KUKA KRL program: MyProgram_163().src

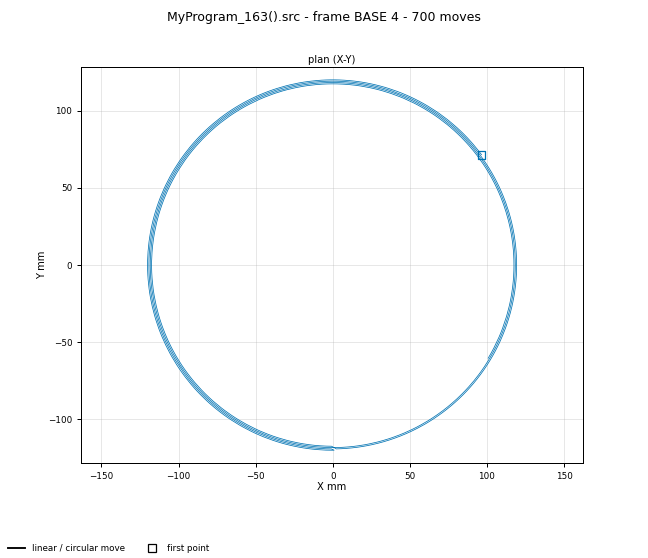
[picture p0: tool path of MyProgram_163().src in frame BASE 4, 700 of 700 moves have a stored position in this frame; points joined in program order, loops and branches not executed]
&ACCESS RVP
&REL 1
&PARAM TEMPLATE = C:\KRC\Roboter\Template\vorgabe
&PARAM EDITMASK = *
DEF MyProgram_163()
; ---- Setting reference (Base) ----
$BASE = BASE_DATA[4]

; --------------------------
; ---- Setting tool (TCP) ----
$TOOL = TOOL_DATA[3]
; --------------------------

$VEL.CP = VEL_APROX_PRINT
Startdeposition()
$VEL.CP = VEL_PRINT
LIN {X 96.4825,Y 71.5563,Z 124,A 32.763,B 24.9424,C -1.7531,E1 25.1279,E2 413.2714} C_DIS
LIN {X 94.5565,Y 74.0809,Z 124,A 34.1726,B 24.9424,C -1.7517,E1 25.1255,E2 411.8718} C_DIS
LIN {X 92.5032,Y 76.6279,Z 124,A 35.5868,B 24.9427,C -1.7484,E1 25.123,E2 410.4719} C_DIS
LIN {X 90.9571,Y 78.4601,Z 124,A 36.9601,B 24.9418,C -1.7622,E1 25.1205,E2 409.0724} C_DIS
LIN {X 89.0042,Y 80.6687,Z 124,A 38.3594,B 24.9416,C -1.7651,E1 25.1179,E2 407.6724} C_DIS
LIN {X 86.9977,Y 82.8287,Z 124,A 39.759,B 24.9414,C -1.7679,E1 25.1152,E2 406.2723} C_DIS
LIN {X 84.9388,Y 84.9388,Z 124,A 41.1588,B 24.9412,C -1.7707,E1 25.1124,E2 404.8719} C_DIS
LIN {X 82.8287,Y 86.9977,Z 124,A 42.5588,B 24.9411,C -1.7733,E1 25.1096,E2 403.4714} C_DIS
LIN {X 80.6687,Y 89.0042,Z 124,A 43.9588,B 24.9409,C -1.7759,E1 25.1067,E2 402.071} C_DIS
LIN {X 78.115,Y 91.2511,Z 124,A 45.38,B 24.9413,C -1.7695,E1 25.1038,E2 400.6704} C_DIS
LIN {X 76.2043,Y 92.8552,Z 124,A 46.7595,B 24.9406,C -1.7809,E1 25.1008,E2 399.2694} C_DIS
LIN {X 73.9026,Y 94.6974,Z 124,A 48.1603,B 24.9404,C -1.7832,E1 25.0977,E2 397.8683} C_DIS
LIN {X 71.2616,Y 96.6983,Z 124,A 49.578,B 24.9407,C -1.7783,E1 25.0946,E2 396.4673} C_DIS
LIN {X 69.167,Y 98.2096,Z 124,A 50.9622,B 24.9401,C -1.7877,E1 25.0914,E2 395.0657} C_DIS
LIN {X 66.736,Y 99.8774,Z 124,A 52.3632,B 24.94,C -1.7898,E1 25.0881,E2 393.6645} C_DIS
LIN {X 63.9427,Y 101.6863,Z 124,A 53.7826,B 24.9403,C -1.7844,E1 25.0849,E2 392.2626} C_DIS
LIN {X 61.7548,Y 103.0317,Z 124,A 55.2287,B 24.9395,C -1.7967,E1 25.0813,E2 390.7918} C_DIS
LIN {X 59.2077,Y 104.5162,Z 124,A 56.5684,B 24.9395,C -1.7956,E1 25.0781,E2 389.4588} C_DIS
LIN {X 56.1374,Y 106.1945,Z 124,A 58.2703,B 24.9393,C -1.7995,E1 25.0739,E2 387.7527} C_DIS
LIN {X 53.3205,Y 107.6363,Z 124,A 59.7249,B 24.9393,C -1.7988,E1 25.0703,E2 386.3035} C_DIS
LIN {X 50.7178,Y 108.8868,Z 124,A 61.1244,B 24.9392,C -1.8015,E1 25.0668,E2 384.9011} C_DIS
LIN {X 47.8151,Y 110.1926,Z 124,A 62.6869,B 24.9389,C -1.8054,E1 25.0628,E2 383.3335} C_DIS
LIN {X 44.6032,Y 111.5336,Z 124,A 64.2825,B 24.9389,C -1.804,E1 25.0586,E2 381.7446} C_DIS
LIN {X 41.8526,Y 112.5946,Z 124,A 65.6861,B 24.9389,C -1.8053,E1 25.055,E2 380.3411} C_DIS
LIN {X 38.6209,Y 113.7415,Z 124,A 67.1118,B 24.9395,C -1.7969,E1 25.0513,E2 378.938} C_DIS
LIN {X 36.2774,Y 114.5126,Z 124,A 68.4935,B 24.9388,C -1.8074,E1 25.0476,E2 377.5341} C_DIS
LIN {X 33.4562,Y 115.3684,Z 124,A 69.8975,B 24.9388,C -1.8084,E1 25.0438,E2 376.1303} C_DIS
LIN {X 30.6149,Y 116.1547,Z 124,A 71.3016,B 24.9386,C -1.8092,E1 25.04,E2 374.7265} C_DIS
LIN {X 27.7551,Y 116.871,Z 124,A 72.706,B 24.9386,C -1.8099,E1 25.0362,E2 373.3223} C_DIS
LIN {X 24.8785,Y 117.517,Z 124,A 74.1109,B 24.9386,C -1.8106,E1 25.0324,E2 371.9177} C_DIS
LIN {X 21.987,Y 118.0921,Z 124,A 75.5159,B 24.9386,C -1.8111,E1 25.0285,E2 370.5132} C_DIS
LIN {X 19.0823,Y 118.5962,Z 124,A 76.9212,B 24.9385,C -1.8116,E1 25.0246,E2 369.1082} C_DIS
LIN {X 16.166,Y 119.0288,Z 124,A 78.3267,B 24.9385,C -1.8119,E1 25.0208,E2 367.7032} C_DIS
LIN {X 13.2401,Y 119.3896,Z 124,A 79.7322,B 24.9385,C -1.8121,E1 25.0169,E2 366.2981} C_DIS
LIN {X 10.3061,Y 119.6786,Z 124,A 81.1409,B 24.9385,C -1.8124,E1 25.0129,E2 364.8897} C_DIS
LIN {X 7.3659,Y 119.8955,Z 124,A 82.5443,B 24.9385,C -1.8123,E1 25.009,E2 363.4871} C_DIS
LIN {X 4.4213,Y 120.0402,Z 124,A 83.951,B 24.9385,C -1.8123,E1 25.0051,E2 362.081} C_DIS
LIN {X 1.4741,Y 120.1125,Z 124,A 85.3576,B 24.9385,C -1.812,E1 25.0012,E2 360.675} C_DIS
LIN {X -1.4741,Y 120.1125,Z 124,A 86.7645,B 24.9385,C -1.8118,E1 24.9973,E2 359.2688} C_DIS
LIN {X -4.4213,Y 120.0402,Z 124,A 88.1715,B 24.9385,C -1.8114,E1 24.9933,E2 357.8624} C_DIS
LIN {X -7.3659,Y 119.8955,Z 124,A 89.579,B 24.9385,C -1.8109,E1 24.9894,E2 356.4557} C_DIS
LIN {X -10.3061,Y 119.6786,Z 124,A 90.9865,B 24.9385,C -1.8103,E1 24.9855,E2 355.0489} C_DIS
LIN {X -13.6363,Y 119.3432,Z 124,A 92.4129,B 24.9391,C -1.8018,E1 24.9816,E2 353.6419} C_DIS
LIN {X -16.166,Y 119.0288,Z 124,A 93.8336,B 24.9386,C -1.8103,E1 24.9776,E2 352.2001} C_DIS
LIN {X -19.0823,Y 118.5962,Z 124,A 95.2109,B 24.9387,C -1.808,E1 24.9738,E2 350.827} C_DIS
LIN {X -21.987,Y 118.0921,Z 124,A 96.6192,B 24.9387,C -1.807,E1 24.9699,E2 349.4196} C_DIS
LIN {X -25.3754,Y 117.4086,Z 124,A 98.0519,B 24.9395,C -1.796,E1 24.9661,E2 348.0114} C_DIS
LIN {X -27.7551,Y 116.8711,Z 124,A 99.4372,B 24.9389,C -1.8048,E1 24.9623,E2 346.6034} C_DIS
LIN {X -30.6149,Y 116.1547,Z 124,A 100.8465,B 24.939,C -1.8035,E1 24.9585,E2 345.1951} C_DIS
LIN {X -33.6095,Y 115.3229,Z 124,A 102.2635,B 24.9393,C -1.799,E1 24.9547,E2 343.7865} C_DIS
LIN {X -36.2774,Y 114.5126,Z 124,A 103.6656,B 24.9393,C -1.8007,E1 24.9509,E2 342.378} C_DIS
LIN {X -39.0768,Y 113.5878,Z 124,A 105.0757,B 24.9393,C -1.7991,E1 24.9472,E2 340.969} C_DIS
LIN {X -41.8526,Y 112.5946,Z 124,A 106.4858,B 24.9394,C -1.7974,E1 24.9435,E2 339.5599} C_DIS
LIN {X -44.6032,Y 111.5336,Z 124,A 107.8963,B 24.9396,C -1.7957,E1 24.9398,E2 338.1506} C_DIS
LIN {X -47.3269,Y 110.4054,Z 124,A 109.3068,B 24.9396,C -1.7938,E1 24.9362,E2 336.7411} C_DIS
LIN {X -50.0222,Y 109.2107,Z 124,A 110.7178,B 24.9398,C -1.7919,E1 24.9326,E2 335.3313} C_DIS
LIN {X -52.6873,Y 107.9502,Z 124,A 112.2257,B 24.9397,C -1.7942,E1 24.9288,E2 333.8142} C_DIS
LIN {X -55.3206,Y 106.6246,Z 124,A 113.6672,B 24.9397,C -1.7934,E1 24.9252,E2 332.3707} C_DIS
LIN {X -57.9207,Y 105.2349,Z 124,A 114.9515,B 24.9402,C -1.7856,E1 24.9221,E2 331.1013} C_DIS
LIN {X -60.4858,Y 103.7818,Z 124,A 116.3632,B 24.9404,C -1.7833,E1 24.9187,E2 329.6908} C_DIS
LIN {X -63.0145,Y 102.2661,Z 124,A 117.775,B 24.9406,C -1.7809,E1 24.9153,E2 328.2803} C_DIS
LIN {X -65.5053,Y 100.6888,Z 124,A 119.1871,B 24.9407,C -1.7785,E1 24.912,E2 326.8695} C_DIS
LIN {X -67.9566,Y 99.0509,Z 124,A 120.5993,B 24.9409,C -1.7759,E1 24.9087,E2 325.4587} C_DIS
LIN {X -70.3669,Y 97.3534,Z 124,A 122.1858,B 24.9406,C -1.7809,E1 24.9051,E2 323.8548} C_DIS
LIN {X -73.2948,Y 95.1658,Z 124,A 123.7761,B 24.9412,C -1.7706,E1 24.9016,E2 322.2833} C_DIS
LIN {X -75.6552,Y 93.3002,Z 124,A 125.192,B 24.9415,C -1.7666,E1 24.8985,E2 320.8717} C_DIS
LIN {X -77.876,Y 91.4547,Z 124,A 126.5891,B 24.9417,C -1.7643,E1 24.8955,E2 319.4745} C_DIS
LIN {X -80.097,Y 89.516,Z 124,A 128.0021,B 24.9419,C -1.7614,E1 24.8926,E2 318.0629} C_DIS
LIN {X -82.2697,Y 87.5234,Z 124,A 129.4156,B 24.9421,C -1.7584,E1 24.8897,E2 316.6508} C_DIS
LIN {X -84.3928,Y 85.478,Z 124,A 130.829,B 24.9423,C -1.7553,E1 24.8869,E2 315.2388} C_DIS
LIN {X -86.4652,Y 83.3812,Z 124,A 132.2427,B 24.9425,C -1.7521,E1 24.8841,E2 313.8266} C_DIS
LIN {X -88.4854,Y 81.2341,Z 124,A 133.67,B 24.9426,C -1.7495,E1 24.8814,E2 312.3993} C_DIS
LIN {X -90.4523,Y 79.0381,Z 124,A 135.0707,B 24.9429,C -1.7456,E1 24.8788,E2 311.0016} C_DIS
LIN {X -92.4035,Y 76.7479,Z 124,A 136.5141,B 24.9431,C -1.7422,E1 24.8762,E2 309.5596} C_DIS
LIN {X -94.2592,Y 74.4571,Z 124,A 137.9284,B 24.9433,C -1.7388,E1 24.8738,E2 308.1468} C_DIS
LIN {X -96.0216,Y 72.1698,Z 124,A 139.3138,B 24.9436,C -1.7354,E1 24.8714,E2 306.7629} C_DIS
LIN {X -97.7639,Y 69.7916,Z 124,A 140.7284,B 24.9438,C -1.7319,E1 24.8691,E2 305.3498} C_DIS
LIN {X -99.4472,Y 67.3714,Z 124,A 142.1433,B 24.944,C -1.7283,E1 24.8669,E2 303.9364} C_DIS
LIN {X -101.1378,Y 64.8058,Z 124,A 143.605,B 24.9443,C -1.724,E1 24.8647,E2 302.4776} C_DIS
LIN {X -102.6662,Y 62.3562,Z 124,A 145.003,B 24.9445,C -1.7209,E1 24.8626,E2 301.0798} C_DIS
LIN {X -104.1641,Y 59.8205,Z 124,A 146.4171,B 24.9447,C -1.7172,E1 24.8606,E2 299.6672} C_DIS
LIN {X -105.6008,Y 57.2461,Z 124,A 147.819,B 24.945,C -1.7129,E1 24.8588,E2 298.2683} C_DIS
LIN {X -107.0122,Y 54.5623,Z 124,A 149.2718,B 24.9453,C -1.7088,E1 24.8569,E2 296.8174} C_DIS
LIN {X -108.2825,Y 51.9956,Z 124,A 150.6629,B 24.9455,C -1.7058,E1 24.8552,E2 295.426} C_DIS
LIN {X -109.5259,Y 49.3226,Z 124,A 152.0655,B 24.9458,C -1.7013,E1 24.8536,E2 294.0263} C_DIS
LIN {X -110.7034,Y 46.6198,Z 124,A 153.4938,B 24.946,C -1.698,E1 24.852,E2 292.5981} C_DIS
LIN {X -111.792,Y 43.9454,Z 124,A 154.8937,B 24.9462,C -1.6946,E1 24.8505,E2 291.1984} C_DIS
LIN {X -112.8576,Y 41.1317,Z 124,A 156.3363,B 24.9464,C -1.6905,E1 24.8491,E2 289.7576} C_DIS
LIN {X -113.8851,Y 38.1951,Z 124,A 157.883,B 24.9466,C -1.6885,E1 24.8477,E2 288.2068} C_DIS
LIN {X -114.9492,Y 34.8694,Z 124,A 159.4964,B 24.9471,C -1.6809,E1 24.8464,E2 286.6022} C_DIS
LIN {X -115.7703,Y 32.0379,Z 124,A 160.9124,B 24.9473,C -1.6768,E1 24.8453,E2 285.1876} C_DIS
LIN {X -116.5217,Y 29.1872,Z 124,A 162.3285,B 24.9476,C -1.6727,E1 24.8444,E2 283.7731} C_DIS
LIN {X -117.2029,Y 26.3188,Z 124,A 163.7444,B 24.9478,C -1.6686,E1 24.8435,E2 282.3587} C_DIS
LIN {X -117.8134,Y 23.4345,Z 124,A 165.1604,B 24.9481,C -1.6645,E1 24.8427,E2 280.9441} C_DIS
LIN {X -118.3531,Y 20.5362,Z 124,A 166.5765,B 24.9483,C -1.6604,E1 24.842,E2 279.5296} C_DIS
LIN {X -118.8214,Y 17.6255,Z 124,A 167.9925,B 24.9486,C -1.6562,E1 24.8414,E2 278.1151} C_DIS
LIN {X -119.2182,Y 14.7042,Z 124,A 169.4089,B 24.9489,C -1.652,E1 24.8409,E2 276.7001} C_DIS
LIN {X -119.5529,Y 11.6682,Z 124,A 170.8298,B 24.9492,C -1.6458,E1 24.8405,E2 275.2856} C_DIS
LIN {X -119.7961,Y 8.8367,Z 124,A 172.241,B 24.9494,C -1.6437,E1 24.8401,E2 273.8709} C_DIS
LIN {X -119.9855,Y 5.6936,Z 124,A 173.6666,B 24.9499,C -1.6356,E1 24.8399,E2 272.4561} C_DIS
LIN {X -120.0854,Y 2.9479,Z 124,A 175.0732,B 24.9499,C -1.6354,E1 24.8399,E2 271.0415} C_DIS
LIN {X -120.1192,Y -0.4835,Z 124,A 176.796,B 24.9499,C -1.6337,E1 24.8398,E2 269.3123} C_DIS
LIN {X -120.0637,Y -3.6544,Z 124,A 178.245,B 24.9505,C -1.6261,E1 24.8398,E2 267.8727} C_DIS
LIN {X -119.9378,Y -6.5998,Z 124,A 179.6742,B 24.9507,C -1.6225,E1 24.8401,E2 266.4435} C_DIS
LIN {X -119.7398,Y -9.5412,Z 124,A -178.9099,B 24.9509,C -1.6184,E1 24.8404,E2 265.0289} C_DIS
LIN {X -119.4632,Y -12.5371,Z 124,A -177.491,B 24.9512,C -1.613,E1 24.8408,E2 263.6141} C_DIS
LIN {X -119.1274,Y -15.4051,Z 124,A -176.0777,B 24.9514,C -1.6101,E1 24.8413,E2 262.1993} C_DIS
LIN {X -118.7042,Y -18.3838,Z 124,A -174.646,B 24.9517,C -1.6054,E1 24.8418,E2 260.7704} C_DIS
LIN {X -118.2172,Y -21.2914,Z 124,A -173.2434,B 24.952,C -1.6008,E1 24.8425,E2 259.3704} C_DIS
LIN {X -117.6591,Y -24.1862,Z 124,A -171.8273,B 24.9522,C -1.5968,E1 24.8433,E2 257.9556} C_DIS
LIN {X -117.0438,Y -27.0074,Z 124,A -170.4277,B 24.9524,C -1.5934,E1 24.8441,E2 256.5557} C_DIS
LIN {X -116.3306,Y -29.9303,Z 124,A -168.996,B 24.9527,C -1.5888,E1 24.8451,E2 255.1266} C_DIS
LIN {X -115.5776,Y -32.7179,Z 124,A -167.5966,B 24.9529,C -1.5855,E1 24.8462,E2 253.7271} C_DIS
LIN {X -114.7398,Y -35.5445,Z 124,A -166.1679,B 24.9531,C -1.5822,E1 24.8473,E2 252.2981} C_DIS
LIN {X -113.8136,Y -38.4071,Z 124,A -164.7495,B 24.9534,C -1.5771,E1 24.8486,E2 250.8836} C_DIS
LIN {X -112.8576,Y -41.1317,Z 124,A -163.3371,B 24.9536,C -1.5745,E1 24.8499,E2 249.4695} C_DIS
LIN {X -111.792,Y -43.9454,Z 124,A -161.9058,B 24.9538,C -1.5701,E1 24.8513,E2 248.0406} C_DIS
LIN {X -110.6798,Y -46.6756,Z 124,A -160.4908,B 24.954,C -1.5663,E1 24.8528,E2 246.6267} C_DIS
LIN {X -109.501,Y -49.3778,Z 124,A -159.089,B 24.9543,C -1.5621,E1 24.8544,E2 245.2274} C_DIS
LIN {X -108.2825,Y -51.9956,Z 124,A -157.69,B 24.9545,C -1.5591,E1 24.8561,E2 243.8278} C_DIS
LIN {X -106.9458,Y -54.6923,Z 124,A -156.2588,B 24.9547,C -1.5548,E1 24.8579,E2 242.3991} C_DIS
LIN {X -105.6008,Y -57.2462,Z 124,A -154.8475,B 24.9548,C -1.5525,E1 24.8598,E2 240.9858} C_DIS
LIN {X -104.1641,Y -59.8205,Z 124,A -153.4461,B 24.9551,C -1.5485,E1 24.8617,E2 239.5868} C_DIS
LIN {X -102.6332,Y -62.4106,Z 124,A -152.0026,B 24.9553,C -1.545,E1 24.8638,E2 238.1441} C_DIS
LIN {X -101.1033,Y -64.8595,Z 124,A -150.6177,B 24.9555,C -1.5417,E1 24.8658,E2 236.7601} C_DIS
LIN {X -99.4472,Y -67.3714,Z 124,A -149.1742,B 24.9557,C -1.5383,E1 24.8681,E2 235.3173} C_DIS
LIN {X -97.6554,Y -69.9437,Z 124,A -147.6122,B 24.9557,C -1.5374,E1 24.8706,E2 233.7498} C_DIS
LIN {X -95.5972,Y -72.7349,Z 124,A -146.0079,B 24.9561,C -1.5311,E1 24.8733,E2 232.1528} C_DIS
LIN {X -93.6748,Y -75.193,Z 124,A -144.5862,B 24.9565,C -1.5246,E1 24.8757,E2 230.7398} C_DIS
LIN {X -91.9131,Y -77.338,Z 124,A -143.1807,B 24.9565,C -1.525,E1 24.8782,E2 229.3269} C_DIS
LIN {X -89.9874,Y -79.5704,Z 124,A -141.7676,B 24.9565,C -1.5221,E1 24.8808,E2 227.9145} C_DIS
LIN {X -88.0076,Y -81.7548,Z 124,A -140.3545,B 24.9568,C -1.5192,E1 24.8835,E2 226.5019} C_DIS
LIN {X -85.9747,Y -83.89,Z 124,A -138.9417,B 24.9569,C -1.5164,E1 24.8862,E2 225.0896} C_DIS
LIN {X -83.8593,Y -86.0043,Z 124,A -137.527,B 24.9571,C -1.5129,E1 24.889,E2 223.6775} C_DIS
LIN {X -81.7548,Y -88.0076,Z 124,A -136.1165,B 24.9572,C -1.5111,E1 24.8919,E2 222.2654} C_DIS
LIN {X -79.5704,Y -89.9874,Z 124,A -134.6582,B 24.9572,C -1.5106,E1 24.895,E2 220.8026} C_DIS
LIN {X -77.338,Y -91.9131,Z 124,A -133.2919,B 24.9575,C -1.5061,E1 24.8979,E2 219.4417} C_DIS
LIN {X -75.0591,Y -93.7834,Z 124,A -131.7279,B 24.9573,C -1.5105,E1 24.9013,E2 217.8614} C_DIS
LIN {X -72.7349,Y -95.5972,Z 124,A -130.4684,B 24.9578,C -1.5014,E1 24.904,E2 216.6189} C_DIS
LIN {X -70.3669,Y -97.3534,Z 124,A -129.057,B 24.9578,C -1.4992,E1 24.9072,E2 215.2078} C_DIS
LIN {X -67.9566,Y -99.0509,Z 124,A -127.4996,B 24.9576,C -1.5036,E1 24.9108,E2 213.6346} C_DIS
LIN {X -65.5053,Y -100.6888,Z 124,A -126.2346,B 24.9581,C -1.495,E1 24.9137,E2 212.386} C_DIS
LIN {X -62.8141,Y -102.3879,Z 124,A -124.8127,B 24.9585,C -1.4884,E1 24.9171,E2 210.9753} C_DIS
LIN {X -60.4858,Y -103.7818,Z 124,A -123.2395,B 24.9579,C -1.499,E1 24.9209,E2 209.3721} C_DIS
LIN {X -57.9207,Y -105.2349,Z 124,A -122.0025,B 24.9584,C -1.4894,E1 24.9239,E2 208.1543} C_DIS
LIN {X -54.8467,Y -106.8669,Z 124,A -120.5673,B 24.9591,C -1.4771,E1 24.9274,E2 206.7443} C_DIS
LIN {X -52.6873,Y -107.9502,Z 124,A -119.1824,B 24.9586,C -1.4861,E1 24.9309,E2 205.3343} C_DIS
LIN {X -50.0222,Y -109.2107,Z 124,A -117.7726,B 24.9587,C -1.4847,E1 24.9345,E2 203.9246} C_DIS
LIN {X -47.3269,Y -110.4054,Z 124,A -116.363,B 24.9587,C -1.4833,E1 24.9381,E2 202.5149} C_DIS
LIN {X -44.6032,Y -111.5336,Z 124,A -114.9061,B 24.9587,C -1.4842,E1 24.9419,E2 201.0526} C_DIS
LIN {X -41.6064,Y -112.6844,Z 124,A -113.5323,B 24.9592,C -1.4756,E1 24.9454,E2 199.6964} C_DIS
LIN {X -39.0768,Y -113.5878,Z 124,A -112.1361,B 24.959,C -1.4797,E1 24.9491,E2 198.2876} C_DIS
LIN {X -36.2774,Y -114.5126,Z 124,A -110.7272,B 24.959,C -1.4787,E1 24.9529,E2 196.8785} C_DIS
LIN {X -33.4562,Y -115.3684,Z 124,A -109.3189,B 24.959,C -1.4778,E1 24.9567,E2 195.47} C_DIS
LIN {X -30.6149,Y -116.1547,Z 124,A -107.9109,B 24.9591,C -1.477,E1 24.9605,E2 194.0618} C_DIS
LIN {X -27.7551,Y -116.8711,Z 124,A -106.502,B 24.9591,C -1.4764,E1 24.9643,E2 192.6524} C_DIS
LIN {X -24.8785,Y -117.517,Z 124,A -105.0952,B 24.9592,C -1.4757,E1 24.9681,E2 191.2455} C_DIS
LIN {X -21.987,Y -118.0921,Z 124,A -103.6879,B 24.9592,C -1.4752,E1 24.972,E2 189.8378} C_DIS
LIN {X -19.0823,Y -118.5962,Z 124,A -102.2806,B 24.9592,C -1.4748,E1 24.9759,E2 188.43} C_DIS
LIN {X -16.166,Y -119.0288,Z 124,A -100.8736,B 24.9592,C -1.4746,E1 24.9798,E2 187.0226} C_DIS
LIN {X -13.2401,Y -119.3896,Z 124,A -99.4671,B 24.9592,C -1.4744,E1 24.9837,E2 185.6156} C_DIS
LIN {X -10.3061,Y -119.6786,Z 124,A -98.0605,B 24.9592,C -1.4743,E1 24.9876,E2 184.2085} C_DIS
LIN {X -7.1561,Y -119.9071,Z 124,A -96.4549,B 24.959,C -1.479,E1 24.9921,E2 182.5913} C_DIS
LIN {X -4.4213,Y -120.0402,Z 124,A -95.2482,B 24.9593,C -1.4744,E1 24.9954,E2 181.395} C_DIS
LIN {X -1.4741,Y -120.1125,Z 124,A -93.8425,B 24.9593,C -1.4746,E1 24.9993,E2 179.9888} C_DIS
LIN {X 0.8495,Y -120.1163,Z 124,A -93.0999,B 24.9602,C -1.4579,E1 25.0013,E2 179.2859} C_DIS
Enddeposition()
LIN {X 0.8495,Y -120.1163,Z 124,A -93.0999,B 24.9602,C -1.4579,E1 25.0013,E2 179.2859} C_DIS
Startdeposition()
$VEL.CP = VEL_PRINT
LIN {X -0.9086,Y -119.2481,Z 124,A -94.2495,B 24.9602,C -1.4589,E1 24.9981,E2 180.4331} C_DIS
LIN {X -4.3095,Y -119.1753,Z 124,A -96.1957,B 24.9609,C -1.4444,E1 24.9926,E2 182.4138} C_DIS
LIN {X -10.5482,Y -118.7847,Z 124,A -98.7422,B 24.9598,C -1.4652,E1 24.9856,E2 184.912} C_DIS
LIN {X -13.5113,Y -118.4841,Z 124,A -100.4433,B 24.9604,C -1.4531,E1 24.9808,E2 186.6429} C_DIS
LIN {X -17.3471,Y -117.9844,Z 124,A -102.2953,B 24.9604,C -1.4538,E1 24.9757,E2 188.4946} C_DIS
LIN {X -21.1648,Y -117.3582,Z 124,A -104.0505,B 24.9601,C -1.4591,E1 24.9709,E2 190.239} C_DIS
LIN {X -24.6012,Y -116.6879,Z 124,A -105.8898,B 24.9605,C -1.4527,E1 24.9658,E2 192.0956} C_DIS
LIN {X -28.42,Y -115.8155,Z 124,A -107.6525,B 24.9601,C -1.4591,E1 24.961,E2 193.8456} C_DIS
LIN {X -31.8672,Y -114.9166,Z 124,A -109.4755,B 24.9603,C -1.4552,E1 24.9561,E2 195.6806} C_DIS
LIN {X -35.357,Y -113.8893,Z 124,A -111.1658,B 24.9601,C -1.459,E1 24.9516,E2 197.3647} C_DIS
LIN {X -38.8928,Y -112.7326,Z 124,A -113.0518,B 24.9603,C -1.4561,E1 24.9466,E2 199.2611} C_DIS
LIN {X -42.3587,Y -111.4749,Z 124,A -115.882,B 24.9627,C -1.4114,E1 24.939,E2 202.2035} C_DIS
LIN {X -49.0255,Y -108.7078,Z 124,A -118.1271,B 24.9596,C -1.4686,E1 24.9335,E2 204.318} C_DIS
LIN {X -51.8005,Y -107.4134,Z 124,A -119.6389,B 24.9596,C -1.4686,E1 24.9297,E2 205.8337} C_DIS
LIN {X -55.2299,Y -105.6915,Z 124,A -121.5594,B 24.9596,C -1.4676,E1 24.9249,E2 207.7618} C_DIS
LIN {X -58.4356,Y -103.9533,Z 124,A -123.338,B 24.9596,C -1.4688,E1 24.9205,E2 209.5426} C_DIS
LIN {X -62.5813,Y -101.5134,Z 124,A -125.6725,B 24.9595,C -1.4712,E1 24.9149,E2 211.8786} C_DIS
LIN {X -65.6775,Y -99.5357,Z 124,A -127.3041,B 24.959,C -1.4799,E1 24.9112,E2 213.4948} C_DIS
LIN {X -68.6467,Y -97.5142,Z 124,A -129.1599,B 24.9591,C -1.4771,E1 24.9069,E2 215.3636} C_DIS
LIN {X -72.1893,Y -94.9214,Z 124,A -131.119,B 24.9586,C -1.4873,E1 24.9025,E2 217.3053} C_DIS
LIN {X -74.6388,Y -93.0068,Z 124,A -133.1968,B 24.9598,C -1.4649,E1 24.8979,E2 219.4442} C_DIS
LIN {X -77.7841,Y -90.3929,Z 124,A -134.4988,B 24.958,C -1.4973,E1 24.8952,E2 220.6742} C_DIS
LIN {X -81.2747,Y -87.2677,Z 124,A -136.942,B 24.9582,C -1.4935,E1 24.8901,E2 223.1362} C_DIS
LIN {X -83.8457,Y -84.7986,Z 124,A -138.6371,B 24.958,C -1.4979,E1 24.8867,E2 224.8279} C_DIS
LIN {X -86.3311,Y -82.2697,Z 124,A -140.4782,B 24.958,C -1.4957,E1 24.8832,E2 226.6822} C_DIS
LIN {X -89.3008,Y -79.0362,Z 124,A -142.4251,B 24.9574,C -1.5075,E1 24.8795,E2 228.6097} C_DIS
LIN {X -91.7598,Y -76.1645,Z 124,A -144.3636,B 24.9574,C -1.5065,E1 24.876,E2 230.5593} C_DIS
LIN {X -94.2396,Y -73.0747,Z 124,A -146.2329,B 24.9571,C -1.5126,E1 24.8728,E2 232.4231} C_DIS
LIN {X -96.7104,Y -69.7738,Z 124,A -148.275,B 24.9571,C -1.5149,E1 24.8694,E2 234.4695} C_DIS
LIN {X -101.6426,Y -62.3693,Z 124,A -152.3443,B 24.9559,C -1.5347,E1 24.8632,E2 238.5119} C_DIS
LIN {X -103.5586,Y -59.1322,Z 124,A -154.3041,B 24.9559,C -1.5332,E1 24.8604,E2 240.4857} C_DIS
LIN {X -105.8623,Y -54.9051,Z 124,A -156.5785,B 24.9555,C -1.5412,E1 24.8574,E2 242.753} C_DIS
LIN {X -107.973,Y -50.6244,Z 124,A -159.2947,B 24.9561,C -1.5299,E1 24.8541,E2 245.5108} C_DIS
LIN {X -109.3185,Y -47.6483,Z 124,A -160.5271,B 24.9551,C -1.5486,E1 24.8528,E2 246.7055} C_DIS
LIN {X -110.7063,Y -44.3336,Z 124,A -162.3317,B 24.955,C -1.5504,E1 24.8508,E2 248.5159} C_DIS
LIN {X -112.0876,Y -40.7099,Z 124,A -164.1388,B 24.9545,C -1.5583,E1 24.8491,E2 250.3143} C_DIS
LIN {X -113.3767,Y -36.9688,Z 124,A -166.0891,B 24.9543,C -1.562,E1 24.8473,E2 252.2669} C_DIS
LIN {X -114.3673,Y -33.7793,Z 124,A -167.594,B 24.9538,C -1.5711,E1 24.8461,E2 253.7589} C_DIS
LIN {X -115.2284,Y -30.7158,Z 124,A -169.5376,B 24.9545,C -1.5585,E1 24.8447,E2 255.7437} C_DIS
LIN {X -116.0384,Y -27.5037,Z 124,A -170.7328,B 24.9532,C -1.5799,E1 24.8439,E2 256.8948} C_DIS
LIN {X -116.7334,Y -24.3797,Z 124,A -172.4192,B 24.9533,C -1.5786,E1 24.8429,E2 258.5944} C_DIS
LIN {X -117.4761,Y -20.5095,Z 124,A -174.4096,B 24.9532,C -1.5805,E1 24.8419,E2 260.592} C_DIS
LIN {X -118.0541,Y -16.8565,Z 124,A -176.0713,B 24.9526,C -1.591,E1 24.8412,E2 262.2385} C_DIS
LIN {X -118.5456,Y -12.9668,Z 124,A -177.9811,B 24.9523,C -1.5959,E1 24.8406,E2 264.148} C_DIS
LIN {X -118.8944,Y -9.2243,Z 124,A -179.662,B 24.9516,C -1.607,E1 24.8402,E2 265.8126} C_DIS
LIN {X -119.1031,Y -5.9771,Z 124,A 178.7165,B 24.9515,C -1.6096,E1 24.8399,E2 267.4376} C_DIS
LIN {X -119.2222,Y -2.6833,Z 124,A 177.0032,B 24.9515,C -1.6094,E1 24.8399,E2 269.1617} C_DIS
LIN {X -119.2486,Y 0.8732,Z 124,A 175.3921,B 24.9509,C -1.619,E1 24.8398,E2 270.7596} C_DIS
LIN {X -119.1841,Y 4.0209,Z 124,A 173.7356,B 24.9509,C -1.618,E1 24.8399,E2 272.4286} C_DIS
LIN {X -118.9864,Y 7.9461,Z 124,A 171.9116,B 24.9504,C -1.6268,E1 24.8402,E2 274.2425} C_DIS
LIN {X -118.7073,Y 11.3863,Z 124,A 170.2503,B 24.9501,C -1.6321,E1 24.8406,E2 275.9012} C_DIS
LIN {X -118.3042,Y 15.0041,Z 124,A 168.4558,B 24.9499,C -1.6359,E1 24.8412,E2 277.6973} C_DIS
LIN {X -117.8441,Y 18.2666,Z 124,A 166.8664,B 24.9496,C -1.6408,E1 24.8419,E2 279.2844} C_DIS
LIN {X -117.0758,Y 22.6755,Z 124,A 164.6811,B 24.9492,C -1.6463,E1 24.843,E2 281.4696} C_DIS
LIN {X -115.8658,Y 28.2138,Z 124,A 162.0185,B 24.9485,C -1.6577,E1 24.8446,E2 284.1209} C_DIS
LIN {X -114.2551,Y 34.1576,Z 124,A 159.137,B 24.9477,C -1.6703,E1 24.8467,E2 286.9889} C_DIS
LIN {X -113.4175,Y 36.8427,Z 124,A 157.6393,B 24.9478,C -1.6685,E1 24.848,E2 288.4995} C_DIS
LIN {X -111.7902,Y 41.5218,Z 124,A 154.9447,B 24.9482,C -1.6629,E1 24.8506,E2 291.2227} C_DIS
LIN {X -109.7259,Y 46.7045,Z 124,A 152.5464,B 24.9469,C -1.6829,E1 24.8531,E2 293.5867} C_DIS
LIN {X -108.22,Y 50.0939,Z 124,A 150.7165,B 24.9467,C -1.6864,E1 24.8552,E2 295.4184} C_DIS
LIN {X -106.7333,Y 53.188,Z 124,A 149.1005,B 24.9463,C -1.6927,E1 24.8572,E2 297.028} C_DIS
LIN {X -104.4869,Y 57.4795,Z 124,A 146.5852,B 24.9463,C -1.6918,E1 24.8605,E2 299.5588} C_DIS
LIN {X -102.5854,Y 60.8043,Z 124,A 144.9339,B 24.9455,C -1.7051,E1 24.8628,E2 301.1871} C_DIS
LIN {X -100.6939,Y 63.8907,Z 124,A 143.0375,B 24.9456,C -1.7035,E1 24.8656,E2 303.0969} C_DIS
LIN {X -98.4349,Y 67.3184,Z 124,A 140.9981,B 24.9454,C -1.7062,E1 24.8688,E2 305.1399} C_DIS
LIN {X -96.4855,Y 70.0832,Z 124,A 139.6672,B 24.9444,C -1.7231,E1 24.8709,E2 306.4372} C_DIS
LIN {X -94.6769,Y 72.5073,Z 124,A 138.035,B 24.9446,C -1.7195,E1 24.8737,E2 308.0857} C_DIS
LIN {X -92.4248,Y 75.357,Z 124,A 136.3123,B 24.9442,C -1.7251,E1 24.8767,E2 309.8032} C_DIS
LIN {X -89.7308,Y 78.5449,Z 124,A 134.356,B 24.9438,C -1.7324,E1 24.8802,E2 311.751} C_DIS
LIN {X -85.7767,Y 82.8449,Z 124,A 131.4879,B 24.9435,C -1.7369,E1 24.8857,E2 314.621} C_DIS
LIN {X -83.1345,Y 85.4975,Z 124,A 129.4443,B 24.9439,C -1.7309,E1 24.8898,E2 316.6874} C_DIS
LIN {X -79.7203,Y 88.6883,Z 124,A 126.9343,B 24.9442,C -1.725,E1 24.895,E2 319.2215} C_DIS
LIN {X -76.7203,Y 91.298,Z 124,A 125.4167,B 24.9429,C -1.7459,E1 24.8982,E2 320.6953} C_DIS
LIN {X -73.8278,Y 93.6502,Z 124,A 123.6934,B 24.9424,C -1.7527,E1 24.9019,E2 322.4088} C_DIS
LIN {X -71.0064,Y 95.8095,Z 124,A 121.2018,B 24.9444,C -1.7231,E1 24.9077,E2 324.9796} C_DIS
LIN {X -66.7964,Y 98.7884,Z 124,A 119.6097,B 24.9416,C -1.7657,E1 24.9111,E2 326.4759} C_DIS
LIN {X -64.418,Y 100.3555,Z 124,A 118.1215,B 24.9417,C -1.7632,E1 24.9146,E2 327.9748} C_DIS
LIN {X -61.4782,Y 102.1842,Z 124,A 116.3527,B 24.9418,C -1.7618,E1 24.9188,E2 329.7525} C_DIS
LIN {X -56.5006,Y 105.0178,Z 124,A 114.0451,B 24.9402,C -1.7858,E1 24.9243,E2 332.0099} C_DIS
LIN {X -51.2487,Y 107.6785,Z 124,A 110.2878,B 24.9426,C -1.7504,E1 24.934,E2 335.8611} C_DIS
LIN {X -47.4136,Y 109.4208,Z 124,A 108.9596,B 24.9404,C -1.7833,E1 24.9372,E2 337.1142} C_DIS
LIN {X -44.8215,Y 110.5077,Z 124,A 107.5114,B 24.9405,C -1.781,E1 24.9409,E2 338.5711} C_DIS
LIN {X -41.7792,Y 111.6944,Z 124,A 105.6075,B 24.9414,C -1.7686,E1 24.946,E2 340.5085} C_DIS
LIN {X -36.7399,Y 113.4508,Z 124,A 103.3352,B 24.9403,C -1.7845,E1 24.9519,E2 342.7475} C_DIS
LIN {X -33.6255,Y 114.4129,Z 124,A 101.8139,B 24.9401,C -1.7882,E1 24.9559,E2 344.2626} C_DIS
LIN {X -29.33,Y 115.5889,Z 124,A 99.4968,B 24.9404,C -1.7826,E1 24.9622,E2 346.5963} C_DIS
LIN {X -25.0419,Y 116.5931,Z 124,A 97.5053,B 24.9399,C -1.79,E1 24.9676,E2 348.5729} C_DIS
LIN {X -21.6386,Y 117.273,Z 124,A 95.7571,B 24.9401,C -1.7878,E1 24.9724,E2 350.3282} C_DIS
LIN {X -18.1261,Y 117.8658,Z 124,A 94.0876,B 24.9399,C -1.7909,E1 24.977,E2 351.9919} C_DIS
LIN {X -14.6574,Y 118.3491,Z 124,A 92.433,B 24.9397,C -1.7931,E1 24.9816,E2 353.6424} C_DIS
LIN {X -11.1145,Y 118.7324,Z 124,A 90.6712,B 24.9398,C -1.7919,E1 24.9865,E2 355.4082} C_DIS
LIN {X -7.9101,Y 118.9888,Z 124,A 89.1459,B 24.9398,C -1.7934,E1 24.9907,E2 356.9305} C_DIS
LIN {X -4.7004,Y 119.1595,Z 124,A 87.514,B 24.9399,C -1.79,E1 24.9953,E2 358.5708} C_DIS
LIN {X -0.8136,Y 119.2486,Z 124,A 85.7804,B 24.9395,C -1.7965,E1 25.0001,E2 360.2892} C_DIS
LIN {X 2.4858,Y 119.2258,Z 124,A 84.201,B 24.9395,C -1.797,E1 25.0045,E2 361.8672} C_DIS
LIN {X 5.7686,Y 119.1136,Z 124,A 82.4794,B 24.9399,C -1.7906,E1 25.0094,E2 363.6034} C_DIS
LIN {X 9.5817,Y 118.8659,Z 124,A 80.7469,B 24.9396,C -1.7952,E1 25.0142,E2 365.3241} C_DIS
LIN {X 13.1484,Y 118.5266,Z 124,A 78.8933,B 24.94,C -1.789,E1 25.0193,E2 367.1913} C_DIS
LIN {X 16.9309,Y 118.0435,Z 124,A 77.2415,B 24.9395,C -1.7967,E1 25.0239,E2 368.8234} C_DIS
LIN {X 20.1074,Y 117.5448,Z 124,A 75.606,B 24.9398,C -1.7921,E1 25.0284,E2 370.4682} C_DIS
LIN {X 23.7661,Y 116.8594,Z 124,A 73.8254,B 24.9398,C -1.7917,E1 25.0333,E2 372.2477} C_DIS
LIN {X 26.7556,Y 116.2112,Z 124,A 72.368,B 24.9398,C -1.7915,E1 25.0372,E2 373.7036} C_DIS
LIN {X 30.2559,Y 115.3509,Z 124,A 70.6234,B 24.94,C -1.7898,E1 25.042,E2 375.4495} C_DIS
LIN {X 33.9813,Y 114.3074,Z 124,A 68.7544,B 24.94,C -1.788,E1 25.047,E2 377.3195} C_DIS
LIN {X 37.6754,Y 113.1444,Z 124,A 66.9235,B 24.94,C -1.7879,E1 25.0518,E2 379.1474} C_DIS
LIN {X 46.3321,Y 109.8828,Z 124,A 62.511,B 24.9403,C -1.7849,E1 25.0634,E2 383.5572} C_DIS
LIN {X 49.6004,Y 108.4488,Z 124,A 60.5576,B 24.9412,C -1.7719,E1 25.0684,E2 385.5365} C_DIS
LIN {X 53.8467,Y 106.4033,Z 124,A 58.505,B 24.9407,C -1.7789,E1 25.0735,E2 387.5673} C_DIS
LIN {X 56.8704,Y 104.8172,Z 124,A 56.8441,B 24.9409,C -1.7757,E1 25.0776,E2 389.2309} C_DIS
LIN {X 60.3043,Y 102.8809,Z 124,A 54.7179,B 24.9418,C -1.7622,E1 25.0828,E2 391.3827} C_DIS
LIN {X 65.142,Y 99.8888,Z 124,A 52.1625,B 24.9415,C -1.7661,E1 25.0887,E2 393.9206} C_DIS
LIN {X 68.939,Y 97.306,Z 124,A 50.0308,B 24.9415,C -1.7658,E1 25.0936,E2 396.0456} C_DIS
LIN {X 71.85,Y 95.1764,Z 124,A 48.3153,B 24.9417,C -1.7636,E1 25.0975,E2 397.7604} C_DIS
LIN {X 75.3333,Y 92.444,Z 124,A 46.3141,B 24.9416,C -1.7655,E1 25.1018,E2 399.7495} C_DIS
LIN {X 77.7251,Y 90.4431,Z 124,A 44.7049,B 24.9421,C -1.7573,E1 25.1053,E2 401.3718} C_DIS
LIN {X 80.568,Y 87.9187,Z 124,A 42.9215,B 24.9422,C -1.7557,E1 25.109,E2 403.152} C_DIS
LIN {X 82.9768,Y 85.6495,Z 124,A 41.3149,B 24.9425,C -1.7515,E1 25.1122,E2 404.7617} C_DIS
LIN {X 85.7538,Y 82.8686,Z 124,A 39.4641,B 24.9427,C -1.7492,E1 25.1158,E2 406.6101} C_DIS
LIN {X 88.1066,Y 80.3633,Z 124,A 37.8299,B 24.9428,C -1.7462,E1 25.1189,E2 408.244} C_DIS
LIN {X 90.5658,Y 77.5811,Z 124,A 35.995,B 24.9433,C -1.7397,E1 25.1223,E2 410.0861} C_DIS
LIN {X 92.9729,Y 74.6806,Z 124,A 34.1423,B 24.9437,C -1.7333,E1 25.1256,E2 411.9453} C_DIS
LIN {X 95.3457,Y 71.6247,Z 124,A 32.3721,B 24.9437,C -1.733,E1 25.1286,E2 413.7079} C_DIS
LIN {X 97.3184,Y 68.9217,Z 124,A 30.7473,B 24.944,C -1.7281,E1 25.1312,E2 415.3363} C_DIS
LIN {X 99.704,Y 65.4224,Z 124,A 28.8504,B 24.944,C -1.7294,E1 25.1342,E2 417.2207} C_DIS
LIN {X 101.4088,Y 62.7488,Z 124,A 27.3133,B 24.9443,C -1.7247,E1 25.1365,E2 418.7611} C_DIS
LIN {X 103.1591,Y 59.8271,Z 124,A 25.2109,B 24.946,C -1.698,E1 25.1395,E2 420.9157} C_DIS
LIN {X 104.9289,Y 56.6645,Z 124,A 24.0193,B 24.9446,C -1.7195,E1 25.141,E2 422.0504} C_DIS
LIN {X 106.2548,Y 54.1372,Z 124,A 22.5575,B 24.9451,C -1.7113,E1 25.1429,E2 423.5239} C_DIS
LIN {X 107.7804,Y 51.0363,Z 124,A 20.7598,B 24.9458,C -1.6999,E1 25.1451,E2 425.3387} C_DIS
LIN {X 109.3702,Y 47.5297,Z 124,A 19.0471,B 24.9458,C -1.7012,E1 25.147,E2 427.0391} C_DIS
LIN {X 110.6013,Y 44.5915,Z 124,A 17.4533,B 24.9462,C -1.6936,E1 25.1487,E2 428.6419} C_DIS
LIN {X 112.2328,Y 40.3117,Z 124,A 15.4009,B 24.9462,C -1.6942,E1 25.1507,E2 430.6815} C_DIS
LIN {X 114.1697,Y 34.4454,Z 124,A 12.2832,B 24.9472,C -1.6779,E1 25.1534,E2 433.82} C_DIS
LIN {X 115.261,Y 30.5952,Z 124,A 10.5534,B 24.947,C -1.6813,E1 25.1547,E2 435.5318} C_DIS
LIN {X 116.0119,Y 27.6151,Z 124,A 8.9666,B 24.9477,C -1.6713,E1 25.1557,E2 437.1329} C_DIS
LIN {X 116.8033,Y 24.0391,Z 124,A 7.2115,B 24.948,C -1.6661,E1 25.1568,E2 438.8902} C_DIS
LIN {X 117.5723,Y 19.9432,Z 124,A 5.2126,B 24.9484,C -1.6599,E1 25.1578,E2 440.8921} C_DIS
LIN {X 118.167,Y 16.0614,Z 124,A 3.3452,B 24.9487,C -1.6547,E1 25.1585,E2 442.7606} C_DIS
LIN {X 118.6062,Y 12.3877,Z 124,A 1.6697,B 24.9487,C -1.654,E1 25.159,E2 444.4279} C_DIS
LIN {X 118.9159,Y 8.9555,Z 124,A -0.1157,B 24.9495,C -1.6423,E1 25.1594,E2 446.2303} C_DIS
LIN {X 119.1517,Y 4.8814,Z 124,A -1.9552,B 24.9495,C -1.6418,E1 25.1597,E2 448.0599} C_DIS
LIN {X 119.2485,Y 0.8916,Z 124,A -3.8677,B 24.9499,C -1.6358,E1 25.1597,E2 449.9752} C_DIS
LIN {X 119.2281,Y -2.3619,Z 124,A -5.4124,B 24.9501,C -1.6316,E1 25.1597,E2 451.5206} C_DIS
LIN {X 119.0784,Y -6.4232,Z 124,A -7.3683,B 24.9505,C -1.6251,E1 25.1595,E2 453.4803} C_DIS
LIN {X 118.8309,Y -10.0193,Z 124,A -9.0056,B 24.9505,C -1.624,E1 25.1591,E2 455.1104} C_DIS
LIN {X 118.515,Y -13.2475,Z 124,A -10.6752,B 24.9512,C -1.6135,E1 25.1587,E2 456.795} C_DIS
LIN {X 118.0446,Y -16.9234,Z 124,A -12.3855,B 24.9514,C -1.6111,E1 25.158,E2 458.5008} C_DIS
LIN {X 117.4661,Y -20.5647,Z 124,A -14.1962,B 24.9518,C -1.6034,E1 25.1572,E2 460.319} C_DIS
LIN {X 116.7758,Y -24.173,Z 124,A -15.8857,B 24.952,C -1.6014,E1 25.1563,E2 462.0035} C_DIS
LIN {X 116.1375,Y -27.0746,Z 124,A -17.299,B 24.9522,C -1.5974,E1 25.1554,E2 463.4178} C_DIS
LIN {X 115.1813,Y -30.8901,Z 124,A -19.2072,B 24.9526,C -1.5904,E1 25.1541,E2 465.3315} C_DIS
LIN {X 114.121,Y -34.6094,Z 124,A -21.0358,B 24.9529,C -1.5859,E1 25.1526,E2 467.1603} C_DIS
LIN {X 112.9916,Y -38.1288,Z 124,A -22.7527,B 24.953,C -1.5832,E1 25.1511,E2 468.8739} C_DIS
LIN {X 111.862,Y -41.3284,Z 124,A -24.6461,B 24.9541,C -1.5652,E1 25.1493,E2 470.7991} C_DIS
LIN {X 110.2446,Y -45.4679,Z 124,A -26.6195,B 24.9541,C -1.5664,E1 25.1473,E2 472.7587} C_DIS
LIN {X 108.3792,Y -49.7518,Z 124,A -28.675,B 24.9539,C -1.5687,E1 25.145,E2 474.7976} C_DIS
LIN {X 107.0576,Y -52.5337,Z 124,A -30.3291,B 24.9547,C -1.5558,E1 25.1429,E2 476.4734} C_DIS
LIN {X 105.4598,Y -55.67,Z 124,A -31.8817,B 24.9546,C -1.5574,E1 25.1409,E2 478.0137} C_DIS
LIN {X 103.9933,Y -58.3639,Z 124,A -33.5643,B 24.9554,C -1.5429,E1 25.1386,E2 479.7218} C_DIS
LIN {X 102.1454,Y -61.542,Z 124,A -35.6215,B 24.9565,C -1.5237,E1 25.1356,E2 481.8138} C_DIS
LIN {X 100.042,Y -64.9064,Z 124,A -37.1246,B 24.9557,C -1.5377,E1 25.1334,E2 483.2765} C_DIS
LIN {X 97.7244,Y -68.3444,Z 124,A -38.9696,B 24.9557,C -1.5392,E1 25.1305,E2 485.1089} C_DIS
LIN {X 95.6996,Y -71.1535,Z 124,A -40.7816,B 24.9563,C -1.5274,E1 25.1275,E2 486.9399} C_DIS
LIN {X 93.3237,Y -74.241,Z 124,A -42.4494,B 24.956,C -1.5322,E1 25.1247,E2 488.5885} C_DIS
LIN {X 91.4614,Y -76.5237,Z 124,A -43.9207,B 24.9564,C -1.5257,E1 25.122,E2 490.0683} C_DIS
LIN {X 89.184,Y -79.1666,Z 124,A -45.6415,B 24.9568,C -1.5192,E1 25.1189,E2 491.7968} C_DIS
LIN {X 86.8441,Y -81.7252,Z 124,A -47.2562,B 24.9568,C -1.5174,E1 25.1158,E2 493.4086} C_DIS
LIN {X 84.5796,Y -84.0674,Z 124,A -48.9243,B 24.9574,C -1.5085,E1 25.1125,E2 495.0905} C_DIS
LIN {X 81.7626,Y -86.8088,Z 124,A -51.0227,B 24.9582,C -1.4939,E1 25.1082,E2 497.2147} C_DIS
LIN {X 79.3885,Y -88.9854,Z 124,A -52.5498,B 24.9583,C -1.4913,E1 25.105,E2 498.742} C_DIS
LIN {X 76.9619,Y -91.0933,Z 124,A -53.6908,B 24.9575,C -1.507,E1 25.1027,E2 499.8414} C_DIS
LIN {X 74.6901,Y -92.9653,Z 124,A -55.1583,B 24.9578,C -1.5013,E1 25.0995,E2 501.3169} C_DIS
LIN {X 72.0623,Y -95.0169,Z 124,A -56.8883,B 24.9583,C -1.4917,E1 25.0956,E2 503.0631} C_DIS
LIN {X 69.1482,Y -97.1568,Z 124,A -58.5471,B 24.9583,C -1.4917,E1 25.0919,E2 504.7159} C_DIS
LIN {X 65.5342,Y -99.6302,Z 124,A -60.5936,B 24.9583,C -1.4903,E1 25.0872,E2 506.7591} C_DIS
LIN {X 62.4579,Y -101.5888,Z 124,A -62.4692,B 24.9589,C -1.481,E1 25.0827,E2 508.6506} C_DIS
LIN {X 59.5492,Y -103.319,Z 124,A -64.754,B 24.9608,C -1.447,E1 25.077,E2 511.0088} C_DIS
LIN {X 54.7994,Y -105.9164,Z 124,A -66.4459,B 24.9587,C -1.4853,E1 25.073,E2 512.6056} C_DIS
LIN {X 50.9246,Y -107.8333,Z 124,A -68.6438,B 24.9592,C -1.4761,E1 25.0675,E2 514.8192} C_DIS
LIN {X 47.835,Y -109.2371,Z 124,A -70.3448,B 24.9595,C -1.4703,E1 25.0631,E2 516.5297} C_DIS
LIN {X 43.8183,Y -110.9094,Z 124,A -72.4044,B 24.9595,C -1.4688,E1 25.0578,E2 518.5883} C_DIS
LIN {X 39.9667,Y -112.3558,Z 124,A -74.3475,B 24.9596,C -1.4677,E1 25.0527,E2 520.53} C_DIS
LIN {X 36.6887,Y -113.4673,Z 124,A -76.0463,B 24.9599,C -1.4639,E1 25.0482,E2 522.2344} C_DIS
LIN {X 32.8877,Y -114.6274,Z 124,A -77.8803,B 24.9598,C -1.4652,E1 25.0433,E2 524.0621} C_DIS
LIN {X 29.325,Y -115.5901,Z 124,A -79.7151,B 24.96,C -1.4605,E1 25.0383,E2 525.9052} C_DIS
LIN {X 25.2015,Y -116.5583,Z 124,A -81.6531,B 24.9599,C -1.4631,E1 25.033,E2 527.8345} C_DIS
LIN {X 22.385,Y -117.1317,Z 124,A -82.9662,B 24.9598,C -1.4651,E1 25.0295,E2 529.1414} C_DIS
LIN {X 19.3571,Y -117.6703,Z 124,A -84.4617,B 24.9598,C -1.4631,E1 25.0253,E2 530.64} C_DIS
LIN {X 16.2187,Y -118.1447,Z 124,A -86.0968,B 24.9602,C -1.4569,E1 25.0208,E2 532.2882} C_DIS
LIN {X 12.4618,Y -118.5985,Z 124,A -87.8375,B 24.9602,C -1.4594,E1 25.016,E2 534.0218} C_DIS
LIN {X 8.9471,Y -118.9166,Z 124,A -89.4952,B 24.9601,C -1.4603,E1 25.0114,E2 535.6765} C_DIS
LIN {X 5.5246,Y -119.124,Z 124,A -91.2508,B 24.9604,C -1.4546,E1 25.0064,E2 537.4448} C_DIS
LIN {X 2.2509,Y -119.2302,Z 124,A -92.7519,B 24.9602,C -1.4575,E1 25.0023,E2 538.9389} C_DIS
LIN {X 2.2509,Y -119.2302,Z 124,A -92.7519,B 24.9602,C -1.4575,E1 25.0023,E2 538.9389} C_DIS
Enddeposition()
LIN {X 0.837,Y -118.3785,Z 124,A -93.3677,B 24.9592,C -1.4755,E1 25.0007,E2 539.5119} C_DIS
Startdeposition()
$VEL.CP = VEL_PRINT
LIN {X 3.2642,Y -118.3391,Z 124,A -91.5416,B 24.9575,C -1.5056,E1 25.006,E2 537.6147} C_DIS
LIN {X 6.5186,Y -118.2039,Z 124,A -89.9979,B 24.9575,C -1.5047,E1 25.0103,E2 536.0737} C_DIS
LIN {X 10.2346,Y -117.942,Z 124,A -88.1229,B 24.9573,C -1.5089,E1 25.0155,E2 534.1897} C_DIS
LIN {X 13.6504,Y -117.5939,Z 124,A -86.5544,B 24.9575,C -1.5056,E1 25.0198,E2 532.6301} C_DIS
LIN {X 16.7886,Y -117.1871,Z 124,A -84.9592,B 24.9573,C -1.5096,E1 25.0243,E2 531.0268} C_DIS
LIN {X 20.6483,Y -116.5693,Z 124,A -83.0979,B 24.9573,C -1.5096,E1 25.0294,E2 529.1674} C_DIS
LIN {X 23.5796,Y -116.0117,Z 124,A -81.7083,B 24.9573,C -1.5083,E1 25.0332,E2 527.7825} C_DIS
LIN {X 29.0926,Y -114.7538,Z 124,A -78.9247,B 24.9571,C -1.5132,E1 25.0408,E2 524.9914} C_DIS
LIN {X 32.3007,Y -113.8917,Z 124,A -77.3337,B 24.9571,C -1.5142,E1 25.0451,E2 523.4006} C_DIS
LIN {X 36.0913,Y -112.7484,Z 124,A -75.4371,B 24.957,C -1.5155,E1 25.0501,E2 521.5043} C_DIS
LIN {X 38.846,Y -111.8293,Z 124,A -73.9842,B 24.9567,C -1.5195,E1 25.054,E2 520.0447} C_DIS
LIN {X 43.305,Y -110.1786,Z 124,A -71.7392,B 24.9567,C -1.52,E1 25.0598,E2 517.8034} C_DIS
LIN {X 46.5749,Y -108.8387,Z 124,A -69.7039,B 24.9557,C -1.538,E1 25.0652,E2 515.7305} C_DIS
LIN {X 51.1975,Y -106.7402,Z 124,A -67.572,B 24.9563,C -1.5264,E1 25.0705,E2 513.6313} C_DIS
LIN {X 54.2782,Y -105.2081,Z 124,A -65.5282,B 24.9551,C -1.5473,E1 25.0757,E2 511.5437} C_DIS
LIN {X 57.3266,Y -103.578,Z 124,A -64.1058,B 24.9557,C -1.5383,E1 25.0791,E2 510.1469} C_DIS
LIN {X 61.2338,Y -101.3171,Z 124,A -62.0491,B 24.9557,C -1.5362,E1 25.084,E2 508.1013} C_DIS
LIN {X 64.2834,Y -99.4105,Z 124,A -60.4159,B 24.9559,C -1.5345,E1 25.0878,E2 506.4776} C_DIS
LIN {X 68.1228,Y -96.8213,Z 124,A -58.0476,B 24.9553,C -1.5451,E1 25.0933,E2 504.0922} C_DIS
LIN {X 71.5775,Y -94.2956,Z 124,A -55.7112,B 24.9543,C -1.5623,E1 25.0986,E2 501.7235} C_DIS
LIN {X 74.1227,Y -92.308,Z 124,A -54.4545,B 24.9549,C -1.551,E1 25.1013,E2 500.4983} C_DIS
LIN {X 77.1784,Y -89.7688,Z 124,A -52.4084,B 24.9543,C -1.5614,E1 25.1057,E2 498.4356} C_DIS
LIN {X 80.6966,Y -86.62,Z 124,A -50.2659,B 24.9544,C -1.5599,E1 25.1101,E2 496.3053} C_DIS
LIN {X 83.939,Y -83.4808,Z 124,A -48.2772,B 24.9547,C -1.5558,E1 25.114,E2 494.3346} C_DIS
LIN {X 86.1077,Y -81.2413,Z 124,A -46.6281,B 24.954,C -1.5664,E1 25.1172,E2 492.6677} C_DIS
LIN {X 88.3807,Y -78.7628,Z 124,A -44.9378,B 24.9536,C -1.5736,E1 25.1204,E2 490.9677} C_DIS
LIN {X 91.6612,Y -74.9208,Z 124,A -42.5578,B 24.9534,C -1.5769,E1 25.1247,E2 488.5908} C_DIS
LIN {X 94.6986,Y -71.041,Z 124,A -40.1793,B 24.953,C -1.5831,E1 25.1287,E2 486.209} C_DIS
LIN {X 96.3847,Y -68.736,Z 124,A -38.4597,B 24.9518,C -1.6035,E1 25.1316,E2 484.4497} C_DIS
LIN {X 98.4134,Y -65.8022,Z 124,A -37.065,B 24.9525,C -1.5921,E1 25.1337,E2 483.0888} C_DIS
LIN {X 100.4759,Y -62.6041,Z 124,A -35.2664,B 24.9523,C -1.5953,E1 25.1364,E2 481.2917} C_DIS
LIN {X 101.7608,Y -60.4936,Z 124,A -33.3913,B 24.9501,C -1.6322,E1 25.1392,E2 479.3392} C_DIS
LIN {X 104.2126,Y -56.1648,Z 124,A -31.6067,B 24.9515,C -1.6087,E1 25.1415,E2 477.6195} C_DIS
LIN {X 106.0596,Y -52.5929,Z 124,A -29.918,B 24.9519,C -1.6019,E1 25.1436,E2 475.9555} C_DIS
LIN {X 108.6963,Y -46.9038,Z 124,A -26.6649,B 24.9507,C -1.6219,E1 25.1474,E2 472.6732} C_DIS
LIN {X 110.1024,Y -43.4991,Z 124,A -25.0725,B 24.9509,C -1.6181,E1 25.149,E2 471.0984} C_DIS
LIN {X 111.9366,Y -38.5401,Z 124,A -22.3797,B 24.9501,C -1.6327,E1 25.1516,E2 468.3864} C_DIS
LIN {X 113.0077,Y -35.27,Z 124,A -20.8098,B 24.9501,C -1.6333,E1 25.1529,E2 466.8239} C_DIS
LIN {X 114.0116,Y -31.8775,Z 124,A -18.6854,B 24.9484,C -1.6591,E1 25.1546,E2 464.651} C_DIS
LIN {X 114.9192,Y -28.4322,Z 124,A -17.3367,B 24.9492,C -1.6461,E1 25.1554,E2 463.3406} C_DIS
LIN {X 115.9397,Y -23.9301,Z 124,A -15.213,B 24.9492,C -1.6479,E1 25.1567,E2 461.2249} C_DIS
LIN {X 116.4895,Y -21.0919,Z 124,A -13.8155,B 24.9488,C -1.6524,E1 25.1574,E2 459.8251} C_DIS
LIN {X 116.9771,Y -18.1943,Z 124,A -12.3943,B 24.9486,C -1.657,E1 25.1581,E2 458.4013} C_DIS
LIN {X 117.5035,Y -14.4225,Z 124,A -10.4421,B 24.9478,C -1.6683,E1 25.1588,E2 456.434} C_DIS
LIN {X 117.8848,Y -10.8551,Z 124,A -8.8134,B 24.9478,C -1.6688,E1 25.1592,E2 454.8139} C_DIS
LIN {X 118.1668,Y -7.1899,Z 124,A -6.9297,B 24.9471,C -1.6797,E1 25.1596,E2 452.9157} C_DIS
LIN {X 118.3293,Y -3.5838,Z 124,A -5.3168,B 24.9471,C -1.6788,E1 25.1597,E2 451.3143} C_DIS
LIN {X 118.3852,Y 0.1464,Z 124,A -3.4385,B 24.9466,C -1.6883,E1 25.1597,E2 449.4249} C_DIS
LIN {X 118.3277,Y 3.6333,Z 124,A -1.8184,B 24.9464,C -1.6905,E1 25.1597,E2 447.8093} C_DIS
LIN {X 118.1403,Y 7.5943,Z 124,A 0.0753,B 24.9461,C -1.6955,E1 25.1594,E2 445.915} C_DIS
LIN {X 117.8999,Y 10.6916,Z 124,A 1.5378,B 24.9459,C -1.6983,E1 25.159,E2 444.4545} C_DIS
LIN {X 117.5705,Y 13.8505,Z 124,A 3.1273,B 24.9455,C -1.7059,E1 25.1585,E2 442.8566} C_DIS
LIN {X 117.032,Y 17.8386,Z 124,A 5.0597,B 24.9451,C -1.7113,E1 25.1578,E2 440.9228} C_DIS
LIN {X 116.4691,Y 21.2052,Z 124,A 6.712,B 24.9448,C -1.7166,E1 25.157,E2 439.2677} C_DIS
LIN {X 115.6916,Y 25.1021,Z 124,A 8.532,B 24.9448,C -1.7176,E1 25.1559,E2 437.4559} C_DIS
LIN {X 115.0435,Y 27.9226,Z 124,A 9.9787,B 24.9443,C -1.7243,E1 25.155,E2 436.002} C_DIS
LIN {X 113.729,Y 32.8749,Z 124,A 12.3727,B 24.9441,C -1.7277,E1 25.1533,E2 433.6135} C_DIS
LIN {X 112.5357,Y 36.7482,Z 124,A 14.6044,B 24.9428,C -1.7469,E1 25.1513,E2 431.3493} C_DIS
LIN {X 111.1972,Y 40.6183,Z 124,A 16.3998,B 24.943,C -1.7437,E1 25.1497,E2 429.5714} C_DIS
LIN {X 109.7653,Y 44.3434,Z 124,A 18.2781,B 24.9428,C -1.7469,E1 25.1477,E2 427.696} C_DIS
LIN {X 108.4316,Y 47.5109,Z 124,A 19.9375,B 24.9425,C -1.7515,E1 25.1459,E2 426.0348} C_DIS
LIN {X 106.3167,Y 52.0743,Z 124,A 22.4076,B 24.9419,C -1.7602,E1 25.143,E2 423.5576} C_DIS
LIN {X 104.6565,Y 55.3327,Z 124,A 23.8564,B 24.9426,C -1.7497,E1 25.1411,E2 422.1412} C_DIS
LIN {X 103.0536,Y 58.2652,Z 124,A 25.9634,B 24.9408,C -1.7778,E1 25.1382,E2 419.979} C_DIS
LIN {X 100.5515,Y 62.483,Z 124,A 28.1027,B 24.9411,C -1.7728,E1 25.1351,E2 417.8622} C_DIS
LIN {X 98.7191,Y 65.3395,Z 124,A 30.3934,B 24.9387,C -1.8085,E1 25.1315,E2 415.4988} C_DIS
LIN {X 95.9081,Y 69.4026,Z 124,A 32.1962,B 24.9402,C -1.786,E1 25.1287,E2 413.7577} C_DIS
LIN {X 91.6726,Y 74.9067,Z 124,A 35.5124,B 24.9398,C -1.7921,E1 25.123,E2 410.4429} C_DIS
LIN {X 89.2143,Y 77.8168,Z 124,A 37.2676,B 24.9398,C -1.7921,E1 25.1198,E2 408.6954} C_DIS
LIN {X 86.6998,Y 80.6116,Z 124,A 39.1678,B 24.9393,C -1.8001,E1 25.1162,E2 406.7848} C_DIS
LIN {X 84.2309,Y 83.1854,Z 124,A 40.7492,B 24.9395,C -1.7971,E1 25.1131,E2 405.2175} C_DIS
LIN {X 82.0197,Y 85.3666,Z 124,A 42.3367,B 24.939,C -1.8043,E1 25.1099,E2 403.6195} C_DIS
LIN {X 79.196,Y 87.9928,Z 124,A 44.1191,B 24.939,C -1.8041,E1 25.1063,E2 401.8447} C_DIS
LIN {X 76.7923,Y 90.0977,Z 124,A 45.7,B 24.9387,C -1.8088,E1 25.1029,E2 400.2589} C_DIS
LIN {X 71.0697,Y 94.6771,Z 124,A 49.1977,B 24.9384,C -1.813,E1 25.0953,E2 396.7643} C_DIS
LIN {X 69.1234,Y 96.1083,Z 124,A 50.8682,B 24.9366,C -1.8387,E1 25.0913,E2 395.0389} C_DIS
LIN {X 65.8766,Y 98.363,Z 124,A 52.4099,B 24.9376,C -1.8243,E1 25.0879,E2 393.5364} C_DIS
LIN {X 62.1217,Y 100.7772,Z 124,A 54.4162,B 24.9379,C -1.8205,E1 25.0831,E2 391.5456} C_DIS
LIN {X 59.2872,Y 102.4686,Z 124,A 55.8218,B 24.9383,C -1.8139,E1 25.0798,E2 390.1599} C_DIS
LIN {X 56.8889,Y 103.8198,Z 124,A 57.3738,B 24.9375,C -1.826,E1 25.076,E2 388.5837} C_DIS
LIN {X 54.0558,Y 105.3217,Z 124,A 58.8998,B 24.9375,C -1.8269,E1 25.0722,E2 387.06} C_DIS
LIN {X 49.2237,Y 107.6666,Z 124,A 61.6205,B 24.9368,C -1.8357,E1 25.0653,E2 384.3255} C_DIS
LIN {X 45.3372,Y 109.3603,Z 124,A 64.071,B 24.9354,C -1.8564,E1 25.0589,E2 381.8317} C_DIS
LIN {X 41.6428,Y 110.818,Z 124,A 65.7434,B 24.9361,C -1.8467,E1 25.0546,E2 380.186} C_DIS
LIN {X 36.8651,Y 112.4981,Z 124,A 67.9286,B 24.9368,C -1.8365,E1 25.0489,E2 378.0291} C_DIS
LIN {X 33.6708,Y 113.4942,Z 124,A 69.542,B 24.9368,C -1.8375,E1 25.0446,E2 376.4163} C_DIS
LIN {X 29.2041,Y 114.7251,Z 124,A 71.7765,B 24.9366,C -1.8386,E1 25.0385,E2 374.1827} C_DIS
LIN {X 25.4781,Y 115.6096,Z 124,A 73.5608,B 24.9368,C -1.8364,E1 25.0337,E2 372.4059} C_DIS
LIN {X 21.2837,Y 116.455,Z 124,A 75.6921,B 24.9365,C -1.84,E1 25.0278,E2 370.2686} C_DIS
LIN {X 17.8553,Y 117.0295,Z 124,A 77.3738,B 24.9365,C -1.8405,E1 25.0232,E2 368.5874} C_DIS
LIN {X 14.0928,Y 117.5421,Z 124,A 79.1973,B 24.9365,C -1.8403,E1 25.0182,E2 366.7659} C_DIS
LIN {X 10.7111,Y 117.8981,Z 124,A 80.8596,B 24.9365,C -1.8413,E1 25.0135,E2 365.1023} C_DIS
LIN {X 6.8181,Y 118.1873,Z 124,A 82.7495,B 24.9365,C -1.8413,E1 25.0083,E2 363.2131} C_DIS
LIN {X 3.5252,Y 118.3311,Z 124,A 84.3381,B 24.9365,C -1.8409,E1 25.0038,E2 361.6259} C_DIS
LIN {X -0.2567,Y 118.3842,Z 124,A 86.22,B 24.9363,C -1.8429,E1 24.9986,E2 359.7395} C_DIS
LIN {X -3.3988,Y 118.3349,Z 124,A 87.7068,B 24.9365,C -1.8409,E1 24.9944,E2 358.2572} C_DIS
LIN {X -6.7696,Y 118.19,Z 124,A 89.3384,B 24.9365,C -1.8403,E1 24.9899,E2 356.6266} C_DIS
LIN {X -10.6244,Y 117.9061,Z 124,A 91.1998,B 24.9366,C -1.839,E1 24.9847,E2 354.7675} C_DIS
LIN {X -13.5416,Y 117.6067,Z 124,A 92.5479,B 24.9369,C -1.8351,E1 24.981,E2 353.4279} C_DIS
LIN {X -17.6299,Y 117.0643,Z 124,A 94.6566,B 24.9366,C -1.8388,E1 24.9751,E2 351.3088} C_DIS
LIN {X -20.6678,Y 116.5658,Z 124,A 96.1411,B 24.9367,C -1.8374,E1 24.9711,E2 349.826} C_DIS
LIN {X -24.3996,Y 115.8433,Z 124,A 98.3622,B 24.9357,C -1.8527,E1 24.9649,E2 347.5659} C_DIS
LIN {X -27.7701,Y 115.0807,Z 124,A 99.6592,B 24.9369,C -1.8346,E1 24.9615,E2 346.3103} C_DIS
LIN {X -36.0869,Y 112.7499,Z 124,A 103.6192,B 24.9379,C -1.8203,E1 24.9509,E2 342.3779} C_DIS
LIN {X -42.1956,Y 110.6086,Z 124,A 106.9836,B 24.9375,C -1.8263,E1 24.942,E2 338.9925} C_DIS
LIN {X -45.822,Y 109.1559,Z 124,A 108.7849,B 24.9379,C -1.8197,E1 24.9374,E2 337.2028} C_DIS
LIN {X -49.4552,Y 107.56,Z 124,A 111.1865,B 24.9367,C -1.8377,E1 24.9312,E2 334.7525} C_DIS
LIN {X -52.528,Y 106.0918,Z 124,A 112.6927,B 24.9373,C -1.8289,E1 24.9274,E2 333.2635} C_DIS
LIN {X -56.4571,Y 104.0541,Z 124,A 114.4071,B 24.9388,C -1.8067,E1 24.9233,E2 331.597} C_DIS
LIN {X -58.6338,Y 102.844,Z 124,A 115.861,B 24.9382,C -1.8153,E1 24.9197,E2 330.1184} C_DIS
LIN {X -62.1442,Y 100.7632,Z 124,A 117.9201,B 24.9382,C -1.8153,E1 24.9148,E2 328.0531} C_DIS
LIN {X -65.2317,Y 98.7901,Z 124,A 119.4535,B 24.9392,C -1.8015,E1 24.9113,E2 326.5474} C_DIS
LIN {X -69.1955,Y 96.0569,Z 124,A 122.0717,B 24.9387,C -1.8091,E1 24.9052,E2 323.9022} C_DIS
LIN {X -72.8659,Y 93.3043,Z 124,A 124.2306,B 24.9392,C -1.8017,E1 24.9004,E2 321.7531} C_DIS
LIN {X -76.1026,Y 90.6829,Z 124,A 126.712,B 24.9381,C -1.8172,E1 24.895,E2 319.2253} C_DIS
LIN {X -79.2118,Y 87.9786,Z 124,A 128.2754,B 24.9397,C -1.7941,E1 24.8919,E2 317.7107} C_DIS
LIN {X -81.365,Y 85.9914,Z 124,A 129.7685,B 24.9397,C -1.7939,E1 24.8888,E2 316.2119} C_DIS
LIN {X -84.2057,Y 83.2109,Z 124,A 131.4776,B 24.9406,C -1.7801,E1 24.8855,E2 314.5285} C_DIS
LIN {X -87.3856,Y 79.8652,Z 124,A 133.8727,B 24.9406,C -1.7813,E1 24.8809,E2 312.12} C_DIS
LIN {X -89.476,Y 77.5172,Z 124,A 135.5818,B 24.9403,C -1.7853,E1 24.8777,E2 310.3937} C_DIS
LIN {X -92.5887,Y 73.7713,Z 124,A 137.7464,B 24.9412,C -1.7708,E1 24.874,E2 308.2534} C_DIS
LIN {X -94.9757,Y 70.6722,Z 124,A 139.7747,B 24.9412,C -1.7714,E1 24.8705,E2 306.214} C_DIS
LIN {X -98.6114,Y 65.5028,Z 124,A 142.7054,B 24.9421,C -1.7574,E1 24.8659,E2 303.3021} C_DIS
LIN {X -100.4966,Y 62.5709,Z 124,A 144.3511,B 24.9425,C -1.7509,E1 24.8635,E2 301.6637} C_DIS
LIN {X -102.1439,Y 59.8455,Z 124,A 145.8927,B 24.9428,C -1.7464,E1 24.8613,E2 300.1248} C_DIS
LIN {X -105.0177,Y 54.6469,Z 124,A 148.9118,B 24.943,C -1.7439,E1 24.8573,E2 297.0957} C_DIS
LIN {X -106.5599,Y 51.5728,Z 124,A 150.4451,B 24.9437,C -1.7334,E1 24.8554,E2 295.5792} C_DIS
LIN {X -107.8486,Y 48.8199,Z 124,A 151.9231,B 24.944,C -1.7292,E1 24.8537,E2 294.1031} C_DIS
LIN {X -109.0463,Y 46.0821,Z 124,A 153.4105,B 24.9441,C -1.7265,E1 24.852,E2 292.6139} C_DIS
LIN {X -110.709,Y 41.9305,Z 124,A 155.7562,B 24.9441,C -1.7273,E1 24.8496,E2 290.253} C_DIS
LIN {X -112.1281,Y 37.9733,Z 124,A 157.5566,B 24.9451,C -1.7111,E1 24.848,E2 288.481} C_DIS
LIN {X -112.9846,Y 35.3444,Z 124,A 158.9612,B 24.9452,C -1.7097,E1 24.8468,E2 287.0718} C_DIS
LIN {X -114.4954,Y 30.0975,Z 124,A 161.7323,B 24.9454,C -1.7066,E1 24.8447,E2 284.2921} C_DIS
LIN {X -115.9593,Y 23.8349,Z 124,A 164.8854,B 24.946,C -1.6982,E1 24.8428,E2 281.1404} C_DIS
LIN {X -117.0917,Y 17.4505,Z 124,A 168.1056,B 24.9464,C -1.6914,E1 24.8413,E2 277.9172} C_DIS
LIN {X -117.6231,Y 13.4014,Z 124,A 169.9115,B 24.9472,C -1.6778,E1 24.8407,E2 276.133} C_DIS
LIN {X -117.9751,Y 9.8328,Z 124,A 171.72,B 24.9474,C -1.6752,E1 24.8402,E2 274.3198} C_DIS
LIN {X -118.1685,Y 7.1581,Z 124,A 173.5108,B 24.9464,C -1.6917,E1 24.84,E2 272.479} C_DIS
LIN {X -118.343,Y 3.1371,Z 124,A 175.0359,B 24.9479,C -1.6675,E1 24.8398,E2 271.0024} C_DIS
LIN {X -118.3816,Y -0.7401,Z 124,A 176.8756,B 24.9484,C -1.6599,E1 24.8398,E2 269.1698} C_DIS
LIN {X -118.2851,Y -4.8322,Z 124,A 179.0451,B 24.9483,C -1.6613,E1 24.84,E2 266.9837} C_DIS
LIN {X -118.0491,Y -8.9073,Z 124,A -178.9124,B 24.9485,C -1.6577,E1 24.8404,E2 264.9375} C_DIS
LIN {X -117.6234,Y -13.3986,Z 124,A -177.0059,B 24.9497,C -1.6391,E1 24.841,E2 263.0641} C_DIS
LIN {X -117.2867,Y -16.0875,Z 124,A -175.3682,B 24.9491,C -1.6486,E1 24.8416,E2 261.3939} C_DIS
LIN {X -115.937,Y -23.9433,Z 124,A -171.7561,B 24.9505,C -1.626,E1 24.8434,E2 257.8143} C_DIS
LIN {X -115.055,Y -27.8754,Z 124,A -169.2146,B 24.9493,C -1.6449,E1 24.8451,E2 255.2128} C_DIS
LIN {X -113.9446,Y -32.1141,Z 124,A -167.6837,B 24.9512,C -1.6134,E1 24.8462,E2 253.7482} C_DIS
LIN {X -113.0213,Y -35.2258,Z 124,A -166.0662,B 24.9514,C -1.6105,E1 24.8475,E2 252.1282} C_DIS
LIN {X -111.7775,Y -38.9934,Z 124,A -164.1304,B 24.9517,C -1.6054,E1 24.8492,E2 250.1936} C_DIS
LIN {X -110.4421,Y -42.6343,Z 124,A -162.1391,B 24.9517,C -1.6046,E1 24.8512,E2 248.1929} C_DIS
LIN {X -109.3471,Y -45.3685,Z 124,A -160.3953,B 24.9512,C -1.614,E1 24.8531,E2 246.4171} C_DIS
LIN {X -107.9292,Y -48.6409,Z 124,A -158.5989,B 24.9513,C -1.612,E1 24.8551,E2 244.6155} C_DIS
LIN {X -106.2287,Y -52.2518,Z 124,A -157.1303,B 24.9528,C -1.5868,E1 24.8569,E2 243.1991} C_DIS
LIN {X -103.6091,Y -57.2719,Z 124,A -154.3229,B 24.9531,C -1.582,E1 24.8606,E2 240.3882} C_DIS
LIN {X -101.8837,Y -60.2858,Z 124,A -152.7186,B 24.9536,C -1.5742,E1 24.8628,E2 238.7942} C_DIS
LIN {X -99.0067,Y -64.903,Z 124,A -149.8192,B 24.9533,C -1.5787,E1 24.8672,E2 235.8694} C_DIS
LIN {X -96.4039,Y -68.7091,Z 124,A -147.798,B 24.9542,C -1.564,E1 24.8704,E2 233.8733} C_DIS
LIN {X -94.5196,Y -71.2794,Z 124,A -146.2641,B 24.9544,C -1.5598,E1 24.8729,E2 232.3421} C_DIS
LIN {X -92.1012,Y -74.3778,Z 124,A -144.3561,B 24.9547,C -1.5554,E1 24.8762,E2 230.4354} C_DIS
LIN {X -90.0927,Y -76.7982,Z 124,A -142.9831,B 24.9553,C -1.5454,E1 24.8787,E2 229.0799} C_DIS
LIN {X -87.2346,Y -80.0299,Z 124,A -140.7082,B 24.9551,C -1.5487,E1 24.883,E2 226.7871} C_DIS
LIN {X -84.5636,Y -82.8485,Z 124,A -138.9917,B 24.9557,C -1.5375,E1 24.8862,E2 225.0898} C_DIS
LIN {X -82.4983,Y -84.9053,Z 124,A -137.3564,B 24.9553,C -1.5442,E1 24.8895,E2 223.4317} C_DIS
LIN {X -80.2288,Y -87.0521,Z 124,A -135.8729,B 24.9556,C -1.5399,E1 24.8926,E2 221.9524} C_DIS
LIN {X -77.6452,Y -89.3643,Z 124,A -133.299,B 24.9535,C -1.5759,E1 24.8982,E2 219.2828} C_DIS
LIN {X -73.1234,Y -93.1008,Z 124,A -131.3983,B 24.9562,C -1.5293,E1 24.9021,E2 217.4858} C_DIS
LIN {X -71.3404,Y -94.4737,Z 124,A -130.0558,B 24.9557,C -1.5384,E1 24.9052,E2 216.1167} C_DIS
LIN {X -67.6994,Y -97.1157,Z 124,A -128.0734,B 24.9564,C -1.5262,E1 24.9096,E2 214.1566} C_DIS
LIN {X -64.6392,Y -99.1808,Z 124,A -126.1895,B 24.9563,C -1.5275,E1 24.914,E2 212.2633} C_DIS
LIN {X -61.7009,Y -101.0332,Z 124,A -124.3409,B 24.956,C -1.5324,E1 24.9185,E2 210.3974} C_DIS
LIN {X -57.6636,Y -103.3904,Z 124,A -122.3376,B 24.9568,C -1.5177,E1 24.9233,E2 208.4231} C_DIS
LIN {X -55.5166,Y -104.5596,Z 124,A -120.7571,B 24.9559,C -1.5338,E1 24.9273,E2 206.8001} C_DIS
LIN {X -52.4629,Y -106.1241,Z 124,A -119.4539,B 24.957,C -1.5158,E1 24.9304,E2 205.5361} C_DIS
LIN {X -48.8205,Y -107.8483,Z 124,A -117.8089,B 24.9579,C -1.4999,E1 24.9345,E2 203.9245} C_DIS
LIN {X -44.5574,Y -109.6782,Z 124,A -114.993,B 24.9565,C -1.523,E1 24.9419,E2 201.0475} C_DIS
LIN {X -40.0762,Y -111.3949,Z 124,A -112.9181,B 24.9573,C -1.5097,E1 24.9473,E2 198.9999} C_DIS
LIN {X -36.6729,Y -112.5603,Z 124,A -111.2233,B 24.9575,C -1.5062,E1 24.9517,E2 197.3101} C_DIS
LIN {X -32.7006,Y -113.7784,Z 124,A -109.1934,B 24.9575,C -1.5056,E1 24.9572,E2 195.2783} C_DIS
LIN {X -29.387,Y -114.6781,Z 124,A -107.5017,B 24.9575,C -1.506,E1 24.9618,E2 193.5832} C_DIS
LIN {X -25.4382,Y -115.6183,Z 124,A -105.6202,B 24.9578,C -1.5012,E1 24.9669,E2 191.7106} C_DIS
LIN {X -22.5399,Y -116.218,Z 124,A -104.1591,B 24.9578,C -1.5019,E1 24.9709,E2 190.2461} C_DIS
LIN {X -19.2488,Y -116.8085,Z 124,A -102.4847,B 24.9576,C -1.504,E1 24.9755,E2 188.5652} C_DIS
LIN {X -15.4082,Y -117.3767,Z 124,A -100.633,B 24.9577,C -1.5023,E1 24.9806,E2 186.716} C_DIS
LIN {X -11.7927,Y -117.7959,Z 124,A -98.7707,B 24.9575,C -1.5067,E1 24.9858,E2 184.8422} C_DIS
LIN {X -8.1368,Y -118.1036,Z 124,A -97.2736,B 24.9582,C -1.4939,E1 24.9899,E2 183.3747} C_DIS
LIN {X -5.9589,Y -118.2347,Z 124,A -95.9834,B 24.9576,C -1.5047,E1 24.9936,E2 182.0587} C_DIS
LIN {X -2.2931,Y -118.3613,Z 124,A -94.268,B 24.9577,C -1.5022,E1 24.9983,E2 180.3489} C_DIS
LIN {X 0.837,Y -118.3785,Z 124,A -93.3655,B 24.9593,C -1.4746,E1 25.0007,E2 179.5119} C_DIS
Enddeposition()
LIN {X 0.837,Y -118.3785,Z 124,A -93.3655,B 24.9593,C -1.4746,E1 25.0007,E2 179.5119} C_DIS
Startdeposition()
$VEL.CP = VEL_PRINT
LIN {X -0.8222,Y -117.5128,Z 124,A -94.2841,B 24.9587,C -1.4847,E1 24.9982,E2 180.4066} C_DIS
LIN {X -4.0859,Y -117.4455,Z 124,A -96.0598,B 24.9592,C -1.4762,E1 24.9932,E2 182.2026} C_DIS
LIN {X -8.0852,Y -117.2373,Z 124,A -97.9058,B 24.9589,C -1.4809,E1 24.988,E2 184.0381} C_DIS
LIN {X -11.739,Y -116.9289,Z 124,A -99.7705,B 24.9591,C -1.4776,E1 24.9828,E2 185.9116} C_DIS
LIN {X -15.315,Y -116.5136,Z 124,A -101.4048,B 24.9588,C -1.4833,E1 24.9783,E2 187.5336} C_DIS
LIN {X -18.9523,Y -115.9781,Z 124,A -103.2726,B 24.9589,C -1.4804,E1 24.9732,E2 189.4099} C_DIS
LIN {X -22.6421,Y -115.3145,Z 124,A -105.1157,B 24.9589,C -1.4804,E1 24.9681,E2 191.2548} C_DIS
LIN {X -26.9414,Y -114.3868,Z 124,A -107.099,B 24.9585,C -1.4886,E1 24.9627,E2 193.2214} C_DIS
LIN {X -29.7962,Y -113.6768,Z 124,A -108.6707,B 24.9588,C -1.4833,E1 24.9584,E2 194.8077} C_DIS
LIN {X -34.982,Y -112.1883,Z 124,A -110.7953,B 24.9574,C -1.5075,E1 24.9529,E2 196.8784} C_DIS
LIN {X -38.4775,Y -111.0388,Z 124,A -112.8779,B 24.9581,C -1.4961,E1 24.9473,E2 198.9919} C_DIS
LIN {X -42.3532,Y -109.6201,Z 124,A -115.8055,B 24.9602,C -1.4583,E1 24.9394,E2 202.0154} C_DIS
LIN {X -46.9332,Y -107.7367,Z 124,A -117.441,B 24.9582,C -1.4945,E1 24.9354,E2 203.5687} C_DIS
LIN {X -49.9063,Y -106.3927,Z 124,A -119.1867,B 24.9584,C -1.4896,E1 24.9309,E2 205.3303} C_DIS
LIN {X -55.9626,Y -103.3349,Z 124,A -122.3906,B 24.9579,C -1.4984,E1 24.923,E2 208.5222} C_DIS
LIN {X -60.7132,Y -100.6179,Z 124,A -124.8653,B 24.9573,C -1.5106,E1 24.9171,E2 210.9753} C_DIS
LIN {X -63.0069,Y -99.1986,Z 124,A -126.4929,B 24.9579,C -1.4991,E1 24.9132,E2 212.6353} C_DIS
LIN {X -66.2347,Y -97.0725,Z 124,A -128.335,B 24.9576,C -1.504,E1 24.9089,E2 214.4718} C_DIS
LIN {X -70.1831,Y -94.2576,Z 124,A -130.5041,B 24.9569,C -1.5164,E1 24.904,E2 216.619} C_DIS
LIN {X -72.126,Y -92.7794,Z 124,A -132.1545,B 24.9579,C -1.499,E1 24.9003,E2 218.3169} C_DIS
LIN {X -77.506,Y -88.3336,Z 124,A -135.1526,B 24.9566,C -1.5227,E1 24.894,E2 221.27} C_DIS
LIN {X -79.6029,Y -86.4485,Z 124,A -136.6028,B 24.9566,C -1.5223,E1 24.891,E2 222.727} C_DIS
LIN {X -82.637,Y -83.5526,Z 124,A -138.6967,B 24.9565,C -1.5245,E1 24.8868,E2 224.8244} C_DIS
LIN {X -85.2421,Y -80.8949,Z 124,A -140.5682,B 24.9564,C -1.5261,E1 24.8831,E2 226.7002} C_DIS
LIN {X -89.4947,Y -76.1618,Z 124,A -143.5556,B 24.9557,C -1.538,E1 24.8776,E2 229.6726} C_DIS
LIN {X -91.3384,Y -73.9406,Z 124,A -145.0672,B 24.9557,C -1.537,E1 24.8749,E2 231.1936} C_DIS
LIN {X -93.9609,Y -70.5781,Z 124,A -147.0366,B 24.9552,C -1.5467,E1 24.8716,E2 233.1494} C_DIS
LIN {X -95.7782,Y -68.0918,Z 124,A -148.6583,B 24.9552,C -1.5454,E1 24.8689,E2 234.7819} C_DIS
LIN {X -97.8257,Y -65.1178,Z 124,A -151.1255,B 24.9567,C -1.5207,E1 24.865,E2 237.3204} C_DIS
LIN {X -100.3843,Y -61.0976,Z 124,A -152.4262,B 24.9539,C -1.5693,E1 24.8632,E2 238.512} C_DIS
LIN {X -101.7629,Y -58.7732,Z 124,A -154.1048,B 24.9545,C -1.5577,E1 24.8608,E2 240.2268} C_DIS
LIN {X -103.972,Y -54.7699,Z 124,A -155.9744,B 24.9533,C -1.5788,E1 24.8583,E2 242.0559} C_DIS
LIN {X -105.2356,Y -52.301,Z 124,A -157.6541,B 24.9539,C -1.569,E1 24.8562,E2 243.7681} C_DIS
LIN {X -106.9024,Y -48.807,Z 124,A -160.1844,B 24.9551,C -1.5479,E1 24.8531,E2 246.3624} C_DIS
LIN {X -108.6316,Y -44.8264,Z 124,A -161.5992,B 24.9531,C -1.5829,E1 24.8517,E2 247.7017} C_DIS
LIN {X -110.3414,Y -40.4317,Z 124,A -164.0401,B 24.953,C -1.5839,E1 24.8492,E2 250.154} C_DIS
LIN {X -111.3499,Y -37.565,Z 124,A -165.4663,B 24.9526,C -1.5907,E1 24.8479,E2 251.5722} C_DIS
LIN {X -112.2757,Y -34.7,Z 124,A -166.9936,B 24.9525,C -1.5927,E1 24.8467,E2 253.1034} C_DIS
LIN {X -113.1868,Y -31.6049,Z 124,A -169.4089,B 24.9542,C -1.5632,E1 24.8448,E2 255.6031} C_DIS
LIN {X -114.5032,Y -26.4375,Z 124,A -170.8267,B 24.9509,C -1.6195,E1 24.8439,E2 256.8948} C_DIS
LIN {X -115.8473,Y -19.7343,Z 124,A -175.1871,B 24.9527,C -1.5881,E1 24.8416,E2 261.356} C_DIS
LIN {X -116.5139,Y -15.313,Z 124,A -176.4793,B 24.9501,C -1.6312,E1 24.8411,E2 262.5531} C_DIS
LIN {X -117.2031,Y -8.5902,Z 124,A -179.9981,B 24.9501,C -1.6326,E1 24.8402,E2 266.0897} C_DIS
LIN {X -117.4211,Y -4.7226,Z 124,A 178.0404,B 24.9499,C -1.6358,E1 24.8399,E2 268.0555} C_DIS
LIN {X -117.5128,Y -0.8684,Z 124,A 176.1014,B 24.9496,C -1.6394,E1 24.8398,E2 269.9973} C_DIS
LIN {X -117.4878,Y 2.5945,Z 124,A 173.5513,B 24.9514,C -1.6101,E1 24.84,E2 272.6327} C_DIS
LIN {X -117.2299,Y 8.1933,Z 124,A 171.7209,B 24.9486,C -1.6555,E1 24.8403,E2 274.366} C_DIS
LIN {X -116.9295,Y 11.7335,Z 124,A 169.8656,B 24.9486,C -1.6561,E1 24.8407,E2 276.231} C_DIS
LIN {X -116.3333,Y 16.628,Z 124,A 167.3354,B 24.9484,C -1.6588,E1 24.8416,E2 278.7698} C_DIS
LIN {X -115.6191,Y 21.0287,Z 124,A 165.3703,B 24.9475,C -1.6744,E1 24.8426,E2 280.7095} C_DIS
LIN {X -114.2146,Y 27.6585,Z 124,A 162.0228,B 24.9469,C -1.6832,E1 24.8446,E2 284.0555} C_DIS
LIN {X -112.8824,Y 32.6791,Z 124,A 159.4967,B 24.9464,C -1.6916,E1 24.8464,E2 286.5765} C_DIS
LIN {X -112.0218,Y 35.5179,Z 124,A 158.0539,B 24.9461,C -1.6963,E1 24.8476,E2 288.0163} C_DIS
LIN {X -110.9518,Y 38.7254,Z 124,A 156.3516,B 24.9459,C -1.6993,E1 24.8491,E2 289.7211} C_DIS
LIN {X -109.6246,Y 42.3404,Z 124,A 154.3574,B 24.9459,C -1.7004,E1 24.8511,E2 291.724} C_DIS
LIN {X -108.3668,Y 45.4597,Z 124,A 152.7492,B 24.9454,C -1.7068,E1 24.8528,E2 293.3259} C_DIS
LIN {X -106.7449,Y 49.1496,Z 124,A 150.7201,B 24.9452,C -1.7101,E1 24.8551,E2 295.3581} C_DIS
LIN {X -105.2823,Y 52.2068,Z 124,A 149.2153,B 24.9445,C -1.7212,E1 24.8569,E2 296.8447} C_DIS
LIN {X -103.9855,Y 54.7442,Z 124,A 147.0631,B 24.9462,C -1.6943,E1 24.8598,E2 299.0725} C_DIS
LIN {X -101.6624,Y 58.9481,Z 124,A 144.8364,B 24.9455,C -1.7058,E1 24.8629,E2 301.2834} C_DIS
LIN {X -99.5215,Y 62.4937,Z 124,A 143.4985,B 24.9433,C -1.7394,E1 24.8648,E2 302.548} C_DIS
LIN {X -95.7502,Y 68.131,Z 124,A 139.7036,B 24.944,C -1.7286,E1 24.8708,E2 306.3874} C_DIS
LIN {X -93.2576,Y 71.5054,Z 124,A 137.9589,B 24.9428,C -1.7465,E1 24.8737,E2 308.0979} C_DIS
LIN {X -91.1291,Y 74.1989,Z 124,A 136.1928,B 24.9428,C -1.7472,E1 24.8768,E2 309.8706} C_DIS
LIN {X -88.4513,Y 77.3712,Z 124,A 134.2258,B 24.9423,C -1.7548,E1 24.8803,E2 311.8284} C_DIS
LIN {X -84.3997,Y 81.7722,Z 124,A 131.2925,B 24.9418,C -1.7614,E1 24.8859,E2 314.7588} C_DIS
LIN {X -81.1886,Y 84.9622,Z 124,A 129.1544,B 24.9413,C -1.7696,E1 24.8902,E2 316.8863} C_DIS
LIN {X -78.604,Y 87.3579,Z 124,A 126.8467,B 24.9427,C -1.7493,E1 24.8951,E2 319.2518} C_DIS
LIN {X -75.5009,Y 90.0544,Z 124,A 125.5083,B 24.9405,C -1.7814,E1 24.8978,E2 320.5189} C_DIS
LIN {X -72.711,Y 92.3205,Z 124,A 123.3306,B 24.9414,C -1.7675,E1 24.9026,E2 322.7377} C_DIS
LIN {X -67.3369,Y 96.3107,Z 124,A 120.2403,B 24.9405,C -1.7815,E1 24.9095,E2 325.8055} C_DIS
LIN {X -64.7261,Y 98.0839,Z 124,A 118.7465,B 24.9402,C -1.7864,E1 24.913,E2 327.2926} C_DIS
LIN {X -60.7152,Y 100.6167,Z 124,A 116.1219,B 24.9408,C -1.7777,E1 24.9193,E2 329.9461} C_DIS
LIN {X -57.8981,Y 102.265,Z 124,A 114.7191,B 24.9401,C -1.7884,E1 24.9226,E2 331.3275} C_DIS
LIN {X -54.5449,Y 104.0905,Z 124,A 113.0235,B 24.9394,C -1.7986,E1 24.9268,E2 333.0037} C_DIS
LIN {X -47.6726,Y 107.4136,Z 124,A 109.3273,B 24.9389,C -1.8055,E1 24.9361,E2 336.6929} C_DIS
LIN {X -44.0521,Y 108.9468,Z 124,A 107.3166,B 24.9389,C -1.8043,E1 24.9413,E2 338.711} C_DIS
LIN {X -38.0265,Y 111.1942,Z 124,A 104.3352,B 24.9383,C -1.8149,E1 24.9491,E2 341.6732} C_DIS
LIN {X -32.9398,Y 112.805,Z 124,A 101.1923,B 24.9396,C -1.7948,E1 24.9576,E2 344.8694} C_DIS
LIN {X -29.6155,Y 113.7233,Z 124,A 100.1002,B 24.9378,C -1.8218,E1 24.9604,E2 345.8991} C_DIS
LIN {X -23.985,Y 115.0425,Z 124,A 97.2815,B 24.9376,C -1.8244,E1 24.968,E2 348.7153} C_DIS
LIN {X -19.6447,Y 115.8623,Z 124,A 94.5378,B 24.9392,C -1.8006,E1 24.9757,E2 351.5183} C_DIS
LIN {X -16.3228,Y 116.3767,Z 124,A 93.4437,B 24.9376,C -1.8252,E1 24.9786,E2 352.5548} C_DIS
LIN {X -13.3414,Y 116.7563,Z 124,A 91.8901,B 24.9378,C -1.8222,E1 24.9829,E2 354.1166} C_DIS
LIN {X -10.7849,Y 117.0197,Z 124,A 90.5406,B 24.938,C -1.8187,E1 24.9867,E2 355.4753} C_DIS
LIN {X -6.8924,Y 117.314,Z 124,A 88.573,B 24.9381,C -1.8166,E1 24.9922,E2 357.4484} C_DIS
LIN {X -3.6243,Y 117.4597,Z 124,A 87.1081,B 24.9377,C -1.8228,E1 24.9962,E2 358.8989} C_DIS
LIN {X -0.5534,Y 117.5144,Z 124,A 85.5904,B 24.9377,C -1.8223,E1 25.0005,E2 360.4178} C_DIS
LIN {X 2.9562,Y 117.4802,Z 124,A 83.7207,B 24.9382,C -1.8156,E1 25.0057,E2 362.3033} C_DIS
LIN {X 6.8893,Y 117.3142,Z 124,A 81.8303,B 24.9382,C -1.8169,E1 25.011,E2 364.1898} C_DIS
LIN {X 11.0924,Y 116.9913,Z 124,A 79.8682,B 24.9379,C -1.8209,E1 25.0164,E2 366.1416} C_DIS
LIN {X 15.0292,Y 116.5506,Z 124,A 77.9255,B 24.9379,C -1.82,E1 25.0218,E2 368.0849} C_DIS
LIN {X 18.0813,Y 116.1163,Z 124,A 76.3647,B 24.9381,C -1.817,E1 25.0261,E2 369.6512} C_DIS
LIN {X 24.4297,Y 114.95,Z 124,A 73.3789,B 24.9377,C -1.8228,E1 25.0343,E2 372.6199} C_DIS
LIN {X 28.5092,Y 114.007,Z 124,A 70.8135,B 24.9394,C -1.7983,E1 25.0414,E2 375.2396} C_DIS
LIN {X 31.9109,Y 113.1001,Z 124,A 69.8447,B 24.9372,C -1.8306,E1 25.0438,E2 376.1304} C_DIS
LIN {X 35.6541,Y 111.9777,Z 124,A 67.7582,B 24.9378,C -1.821,E1 25.0494,E2 378.2359} C_DIS
LIN {X 37.9982,Y 111.2038,Z 124,A 66.4207,B 24.9383,C -1.8139,E1 25.053,E2 379.5876} C_DIS
LIN {X 44.2326,Y 108.8733,Z 124,A 63.5236,B 24.9375,C -1.8265,E1 25.0605,E2 382.4486} C_DIS
LIN {X 46.3339,Y 107.998,Z 124,A 61.9676,B 24.9389,C -1.805,E1 25.0646,E2 384.0518} C_DIS
LIN {X 52.6869,Y 105.0444,Z 124,A 58.7446,B 24.9386,C -1.8096,E1 25.0727,E2 387.2557} C_DIS
LIN {X 55.1829,Y 103.7545,Z 124,A 57.0334,B 24.9398,C -1.7922,E1 25.077,E2 389.0031} C_DIS
LIN {X 59.3324,Y 101.439,Z 124,A 54.8414,B 24.9396,C -1.7946,E1 25.0823,E2 391.183} C_DIS
LIN {X 62.2578,Y 99.6689,Z 124,A 53.3139,B 24.9394,C -1.7984,E1 25.0859,E2 392.6967} C_DIS
LIN {X 65.6274,Y 97.4837,Z 124,A 50.8587,B 24.9411,C -1.7725,E1 25.0917,E2 395.205} C_DIS
LIN {X 69.0074,Y 95.1219,Z 124,A 49.5266,B 24.9393,C -1.8,E1 25.0946,E2 396.4672} C_DIS
LIN {X 74.1594,Y 91.1611,Z 124,A 46.456,B 24.9393,C -1.7987,E1 25.1014,E2 399.5296} C_DIS
LIN {X 76.2503,Y 89.4193,Z 124,A 44.9049,B 24.9402,C -1.7857,E1 25.1047,E2 401.1054} C_DIS
LIN {X 78.7633,Y 87.2154,Z 124,A 43.169,B 24.9408,C -1.7775,E1 25.1083,E2 402.8539} C_DIS
LIN {X 81.5563,Y 84.6079,Z 124,A 41.4698,B 24.9405,C -1.7812,E1 25.1118,E2 404.5373} C_DIS
LIN {X 83.8637,Y 82.3221,Z 124,A 39.7693,B 24.9411,C -1.7723,E1 25.1151,E2 406.2516} C_DIS
LIN {X 86.5344,Y 79.5093,Z 124,A 37.9965,B 24.9411,C -1.7736,E1 25.1185,E2 408.0136} C_DIS
LIN {X 88.5953,Y 77.2062,Z 124,A 36.4578,B 24.9414,C -1.7686,E1 25.1214,E2 409.5571} C_DIS
LIN {X 91.1775,Y 74.1392,Z 124,A 34.0351,B 24.9431,C -1.7422,E1 25.1257,E2 412.0311} C_DIS
LIN {X 93.6373,Y 71.0089,Z 124,A 32.7299,B 24.9415,C -1.767,E1 25.1279,E2 413.2714} C_DIS
LIN {X 97.4447,Y 65.6849,Z 124,A 29.5125,B 24.9421,C -1.7577,E1 25.1331,E2 416.4952} C_DIS
LIN {X 98.8865,Y 63.4931,Z 124,A 28.1246,B 24.9427,C -1.7492,E1 25.1352,E2 417.8962} C_DIS
LIN {X 100.955,Y 60.1513,Z 124,A 25.7386,B 24.9444,C -1.722,E1 25.1387,E2 420.3342} C_DIS
LIN {X 102.9462,Y 56.6766,Z 124,A 24.3912,B 24.9429,C -1.7451,E1 25.1405,E2 421.6202} C_DIS
LIN {X 104.8158,Y 53.1386,Z 124,A 21.9357,B 24.9448,C -1.7158,E1 25.1437,E2 424.1317} C_DIS
LIN {X 106.4026,Y 49.885,Z 124,A 20.8356,B 24.9431,C -1.7422,E1 25.1449,E2 425.1636} C_DIS
LIN {X 107.5625,Y 47.3328,Z 124,A 19.1887,B 24.9442,C -1.7249,E1 25.1468,E2 426.8423} C_DIS
LIN {X 108.8811,Y 44.2135,Z 124,A 17.6528,B 24.9442,C -1.7255,E1 25.1485,E2 428.3683} C_DIS
LIN {X 110.0937,Y 41.1048,Z 124,A 16.0611,B 24.9444,C -1.7224,E1 25.15,E2 429.9586} C_DIS
LIN {X 111.0921,Y 38.3257,Z 124,A 14.0042,B 24.9466,C -1.6888,E1 25.152,E2 432.0831} C_DIS
LIN {X 112.3885,Y 34.3364,Z 124,A 12.6399,B 24.9449,C -1.7148,E1 25.1531,E2 433.3782} C_DIS
LIN {X 113.8649,Y 29.0645,Z 124,A 10.3322,B 24.9443,C -1.7239,E1 25.1548,E2 435.6514} C_DIS
LIN {X 114.8442,Y 24.9147,Z 124,A 7.822,B 24.9461,C -1.6967,E1 25.1564,E2 438.2112} C_DIS
LIN {X 115.5951,Y 21.162,Z 124,A 5.8633,B 24.9467,C -1.6863,E1 25.1574,E2 440.1828} C_DIS
LIN {X 116.1909,Y 17.5987,Z 124,A 4.108,B 24.947,C -1.681,E1 25.1582,E2 441.9403} C_DIS
LIN {X 116.7142,Y 13.7008,Z 124,A 2.2919,B 24.9471,C -1.6797,E1 25.1588,E2 443.7489} C_DIS
LIN {X 117.1018,Y 9.8665,Z 124,A 0.376,B 24.9476,C -1.6718,E1 25.1593,E2 445.6718} C_DIS
LIN {X 117.3371,Y 6.4745,Z 124,A -1.1783,B 24.9476,C -1.6714,E1 25.1596,E2 447.2179} C_DIS
LIN {X 117.4715,Y 3.2392,Z 124,A -2.8337,B 24.9482,C -1.6626,E1 25.1598,E2 448.8842} C_DIS
LIN {X 117.5137,Y -0.7385,Z 124,A -4.6554,B 24.9482,C -1.6619,E1 25.1598,E2 450.6968} C_DIS
LIN {X 117.4624,Y -3.5382,Z 124,A -6.0132,B 24.9485,C -1.6578,E1 25.1597,E2 452.0561} C_DIS
LIN {X 117.3102,Y -6.9622,Z 124,A -7.8008,B 24.9492,C -1.6467,E1 25.1594,E2 453.8592} C_DIS
LIN {X 117.0231,Y -10.7476,Z 124,A -9.5782,B 24.9493,C -1.6442,E1 25.159,E2 455.632} C_DIS
LIN {X 116.598,Y -14.6636,Z 124,A -11.6589,B 24.9502,C -1.6303,E1 25.1583,E2 457.7333} C_DIS
LIN {X 115.8763,Y -19.5612,Z 124,A -13.8518,B 24.95,C -1.633,E1 25.1574,E2 459.9069} C_DIS
LIN {X 115.2228,Y -23.1065,Z 124,A -16.0433,B 24.9516,C -1.6065,E1 25.1562,E2 462.148} C_DIS
LIN {X 114.4545,Y -26.6482,Z 124,A -17.3061,B 24.9505,C -1.6249,E1 25.1554,E2 463.3601} C_DIS
LIN {X 112.7056,Y -33.2773,Z 124,A -20.3762,B 24.9504,C -1.6272,E1 25.1533,E2 466.407} C_DIS
LIN {X 110.1159,Y -41.046,Z 124,A -24.5628,B 24.9517,C -1.6052,E1 25.1495,E2 470.622} C_DIS
LIN {X 109.1295,Y -43.602,Z 124,A -25.9169,B 24.952,C -1.6001,E1 25.1481,E2 471.9805} C_DIS
LIN {X 107.8587,Y -46.6534,Z 124,A -28.9016,B 24.9561,C -1.5302,E1 25.1446,E2 475.1138} C_DIS
LIN {X 104.5556,Y -53.6477,Z 124,A -31.844,B 24.9545,C -1.5578,E1 25.141,E2 477.9756} C_DIS
LIN {X 102.6362,Y -57.234,Z 124,A -33.705,B 24.9545,C -1.5577,E1 25.1385,E2 479.827} C_DIS
LIN {X 100.7839,Y -60.4401,Z 124,A -35.0197,B 24.9535,C -1.5757,E1 25.1367,E2 481.0925} C_DIS
Enddeposition()
END
